Yaskawa INFORM job: SKRZYNIA_4840_-90_STOPNI_10BR.JBI

/JOB
//NAME SKRZYNIA_4840_-90_STOPNI_10BR
///FOLDERNAME 02-SKRZYNIE_JOBS
//POS
///NPOS 688,688,0,49,0,0
///TOOL 0
///POSTYPE PULSE
///PULSE
C00000=0,-52280,40443,0,6876,0
C00001=-82314,-24956,17040,-59626,-27382,-6248
C00002=-93910,-8625,17040,-59626,-43355,-6248
C00003=-98846,-1061,-42166,-80308,-57081,16120
C00004=-100452,6057,-48127,-85711,-56704,21322
C00005=-96957,25597,-37888,-85158,-62082,25522
C00006=-95580,33075,-33256,-84644,-64024,26851
C00007=-94380,33739,-32188,-85134,-63496,26721
C00008=-95580,33075,-33256,-84644,-64024,26851
C00009=-94940,31262,-36138,-85248,-63712,27160
C00010=-95580,33075,-33256,-84644,-64024,26851
C00011=-95263,33142,-33256,-84677,-63995,26850
C00012=-95263,33142,-33256,-84677,-63995,26850
C00013=-94261,33702,-32359,-85087,-63552,26740
C00014=-95263,33142,-33256,-84677,-63995,26850
C00015=-94777,31773,-35433,-85135,-63758,27084
C00016=-95263,33142,-33256,-84677,-63995,26850
C00017=-95260,33144,-33256,-84678,-63995,26850
C00018=-95260,33144,-33256,-84678,-63995,26850
C00019=-94282,33689,-32380,-85076,-63563,26742
C00020=-95260,33144,-33256,-84678,-63995,26850
C00021=-94827,31920,-35204,-85086,-63784,27059
C00022=-95260,33144,-33256,-84678,-63995,26850
C00023=-95258,33145,-33257,-84676,-63996,26846
C00024=-95258,33145,-33257,-84676,-63996,26846
C00025=-94286,33686,-32387,-85074,-63568,26738
C00026=-95258,33145,-33257,-84676,-63996,26846
C00027=-94874,32057,-34990,-85039,-63809,27032
C00028=-95258,33145,-33257,-84676,-63996,26846
C00029=-95258,33145,-33257,-84676,-63996,26846
C00030=-95258,33145,-33257,-84676,-63996,26846
C00031=-94323,33667,-32422,-85059,-63584,26741
C00032=-95258,33145,-33257,-84676,-63996,26846
C00033=-94899,32130,-34875,-85014,-63820,27019
C00034=-95258,33145,-33257,-84676,-63996,26846
C00035=-95258,25631,32269,-66559,-75499,2416
C00036=-95258,25631,32269,-66559,-75499,2416
C00037=-94333,26371,33350,-66433,-74983,2224
C00038=-95258,25631,32269,-66559,-75499,2416
C00039=-94886,24142,30119,-66602,-75133,2534
C00040=-95258,25631,32269,-66559,-75499,2416
C00041=-98646,19496,-17631,-99827,-80462,21224
C00042=-98811,21047,-15512,-99242,-81394,20987
C00043=-97886,21574,-14788,-99528,-80824,20997
C00044=-98811,21047,-15512,-99242,-81394,20987
C00045=-98517,19954,-17009,-99363,-81263,21101
C00046=-98811,21047,-15512,-99242,-81394,20987
C00047=-98811,19937,1242,-97498,-78933,15296
C00048=-98811,19937,1242,-97498,-78933,15296
C00049=-97933,20465,1962,-97646,-78345,15298
C00050=-98811,19937,1242,-97498,-78933,15296
C00051=-98523,18806,-285,-97586,-78782,15407
C00052=-98811,19937,1242,-97498,-78933,15296
C00053=-98215,26829,34899,-99955,-75775,7961
C00054=-97536,27946,37844,-102629,-75095,7996
C00055=-96676,28621,38852,-102572,-74482,7985
C00056=-97536,27946,37844,-102629,-75095,7996
C00057=-97073,25840,34734,-102750,-74944,8293
C00058=-97536,27946,37844,-102629,-75095,7996
C00059=-96761,21976,18943,-104804,-75068,12116
C00060=-92262,-3556,-2957,-107669,-51219,12798
C00061=-85502,-24407,-19904,-109451,-30096,13932
C00062=-50003,-39410,-5978,-16260,-18649,-25999
C00063=-48287,-44591,-17414,-16172,-14532,-25809
C00064=-85348,-13130,13838,-41209,-47455,-8220
C00065=-99199,18818,35660,-68259,-73735,6208
C00066=-95720,15423,18785,-70454,-68603,10022
C00067=-95720,15423,18785,-70454,-68603,10022
C00068=-97322,30100,38585,-71742,-79662,10416
C00069=-96349,30901,39804,-71630,-79090,10224
C00070=-97322,30100,38585,-71742,-79662,10416
C00071=-97054,28837,36680,-71776,-79387,10556
C00072=-97322,30100,38585,-71742,-79662,10416
C00073=-97373,30352,38967,-71736,-79717,10385
C00074=-97373,30352,38967,-71736,-79717,10385
C00075=-96432,31128,40151,-71627,-79165,10198
C00076=-97373,30352,38967,-71736,-79717,10385
C00077=-97071,28917,36802,-71776,-79407,10544
C00078=-97373,30352,38967,-71736,-79717,10385
C00079=-97356,30262,38827,-71739,-79698,10398
C00080=-97356,30262,38827,-71739,-79698,10398
C00081=-96507,30957,39891,-71642,-79201,10230
C00082=-97356,30262,38827,-71739,-79698,10398
C00083=-97092,29010,36937,-71773,-79425,10538
C00084=-97356,30262,38827,-71739,-79698,10398
C00085=-97431,30641,39402,-71725,-79780,10352
C00086=-97431,30641,39402,-71725,-79780,10352
C00087=-96578,31348,40481,-71627,-79280,10181
C00088=-97431,30641,39402,-71725,-79780,10352
C00089=-97114,29116,37095,-71767,-79448,10523
C00090=-97431,30641,39402,-71725,-79780,10352
C00091=-99948,24360,13310,-86634,-79084,-1692
C00092=-99948,24360,13310,-86634,-79084,-1692
C00093=-99080,24906,14086,-86708,-78501,-1755
C00094=-99948,24360,13310,-86634,-79084,-1692
C00095=-99633,22968,11346,-86719,-78869,-1551
C00096=-99948,24360,13310,-86634,-79084,-1692
C00097=-97019,23700,25794,-103927,-75007,-5801
C00098=-97395,30282,35552,-103352,-78262,-7023
C00099=-96588,30934,36542,-103330,-77681,-7037
C00100=-97395,30282,35552,-103352,-78262,-7023
C00101=-97049,28659,33116,-103437,-78167,-6786
C00102=-97395,30282,35552,-103352,-78262,-7023
C00103=-90014,-10558,-39023,-122472,-57861,10563
C00104=-96923,-13864,-45757,-120418,-62715,10144
C00105=-81853,-22326,-62247,-144804,-57102,19611
C00106=-90840,-27079,-68635,-139700,-60795,17408
C00107=-59535,-63832,-86313,-155973,-37716,23892
C00108=-73187,-23116,26488,-26118,-57509,-28469
C00109=-99665,-12992,-24886,-73613,-54905,-950
C00110=-98398,-8109,-25057,-81551,-55130,4513
C00111=-99451,17861,2757,-80571,-73406,6045
C00112=-99056,24650,11359,-80216,-77425,5946
C00113=-98115,25261,12228,-80295,-76818,5843
C00114=-99056,24650,11359,-80216,-77425,5946
C00115=-98800,23560,9817,-80291,-77224,6050
C00116=-99056,24650,11359,-80216,-77425,5946
C00117=-99819,33446,48735,-87787,-79679,-1235
C00118=-99819,33446,48735,-87787,-79679,-1235
C00119=-98945,34179,49898,-87659,-79086,-1350
C00120=-99819,33446,48735,-87787,-79679,-1235
C00121=-99591,32133,46677,-87830,-79529,-1033
C00122=-99819,33446,48735,-87787,-79679,-1235
C00123=-98853,28116,28355,-96898,-79749,4777
C00124=-98853,30464,37910,-96149,-78952,2546
C00125=-98284,30904,38579,-96116,-78548,2515
C00126=-98853,30464,37910,-96149,-78952,2546
C00127=-98656,29478,36421,-96191,-78865,2688
C00128=-98853,30464,37910,-96149,-78952,2546
C00129=-94437,3365,15121,-90804,-55123,21
C00130=-76606,-19838,2636,-59027,-23020,-13375
C00131=-49667,-45532,-21960,-5654,-17518,-35856
C00132=-47485,-50287,-32535,-1070,-13732,-37871
C00133=-36103,-65917,11738,-26975,4295,7905
C00134=6327,-52297,40484,-8600,6957,5944
C00135=0,-43112,23163,32261,-40956,29092
C00136=-48283,-21883,28214,-25170,-26491,48363
C00137=-46664,-3144,58041,-18842,-32105,45325
C00138=-50347,-18571,12268,-49104,-16423,60029
C00139=-53571,-17125,12073,-56866,-17385,63433
C00140=-52069,-15730,13206,-55612,-16432,62999
C00141=-53474,-15384,13495,-57637,-17161,63825
C00142=-53571,-17125,12073,-56866,-17385,63433
C00143=-50509,-19000,10610,-51503,-15997,61182
C00144=-53130,-17211,12007,-56251,-17152,63186
C00145=-51822,-15992,12994,-55136,-16324,62798
C00146=-53635,-15431,13457,-57815,-17251,63894
C00147=-53130,-17211,12007,-56251,-17152,63186
C00148=-50704,-18403,11069,-52157,-16018,61478
C00149=-53231,-16470,14622,-53206,-17893,61673
C00150=-51756,-15101,15744,-51790,-16990,61165
C00151=-53741,-14453,16285,-54808,-17949,62397
C00152=-53231,-17580,11714,-56182,-17246,63139
C00153=-51814,-19410,10295,-53186,-16720,61844
C00154=-53629,-18979,7405,-62018,-16535,65958
C00155=-52238,-17698,8415,-61175,-15613,65699
C00156=-53551,-17401,8655,-62910,-16346,66402
C00157=-52880,-17654,11656,-55678,-17066,62935
C00158=-51005,-17995,11387,-52847,-16122,61778
C00159=-52964,-17611,11689,-55811,-17106,62990
C00160=-51611,-16353,12697,-54642,-16249,62582
C00161=-53495,-15765,13180,-57466,-17201,63739
C00162=-52964,-17611,11689,-55811,-17106,62990
C00163=-51030,-17982,11395,-52891,-16135,61798
C00164=-52975,-17563,11726,-55850,-17109,63009
C00165=-51607,-16289,12749,-54669,-16241,62596
C00166=-53283,-15811,13140,-57177,-17094,63622
C00167=-52975,-17563,11726,-55850,-17109,63009
C00168=-50945,-18019,11363,-52741,-16103,61737
C00169=-52728,-17788,11545,-55393,-17010,62816
C00170=-51045,-16207,12813,-53894,-15944,62287
C00171=-52895,-15647,13274,-56746,-16874,63461
C00172=-52728,-17788,11545,-55393,-17010,62816
C00173=-50945,-18019,11363,-52741,-16103,61737
C00174=-52556,-17520,11756,-55311,-16888,62798
C00175=-51113,-16157,12849,-54025,-15975,62343
C00176=-52730,-15718,13210,-56498,-16792,63358
C00177=-52556,-17520,11756,-55311,-16888,62798
C00178=-50945,-18019,11363,-52741,-16103,61737
C00179=-51893,-17787,11546,-54246,-16568,62356
C00180=-50379,-16341,12703,-52826,-15610,61849
C00181=-52406,-15704,13225,-56071,-16614,63190
C00182=-51893,-17787,11546,-54246,-16568,62356
C00183=-50028,-22953,-3957,-22347,-31919,54220
C00184=-50947,-22502,-3625,-23433,-32061,54736
C00185=-49421,-20951,-2455,-21951,-31329,54057
C00186=-51207,-20433,-2055,-24026,-31698,55041
C00187=-50529,-22709,-3778,-22940,-31995,54502
C00188=-49763,-25421,-36239,-24565,-26935,60445
C00189=-49763,-25421,-36239,-24565,-26935,60445
C00190=-48299,-23485,-34758,-23276,-26122,59713
C00191=-50218,-22723,-34165,-25568,-26529,60993
C00192=-49763,-25421,-36239,-24565,-26935,60445
C00193=-50713,-12366,-58367,-41124,-17813,74400
C00194=-50824,-12254,-58263,-41255,-17847,74484
C00195=-49431,-10052,-56192,-40383,-17131,73813
C00196=-50915,-9358,-55524,-41955,-17664,74847
C00197=-51028,-12852,-58814,-41301,-17980,74542
C00198=-49763,-25421,-36239,-24565,-26935,60445
C00199=-50529,-22709,-3778,-22940,-31995,54502
C00200=-45389,-28224,4312,-35967,-15579,54278
C00201=-40154,-51179,-915,-24203,-8234,36524
C00202=0,-52280,40443,0,6876,0
C00203=0,-52280,40443,0,6876,0
C00204=-2117,-50103,-33543,-4117,45077,85249
C00205=26439,-48928,-33543,-4117,-52362,85249
C00206=26439,-27355,-33543,-41485,-52362,85249
C00207=39218,-24492,-41653,-51934,-39374,86964
C00208=39218,-24492,-41653,-51934,-39374,86964
C00209=46639,7575,-9331,-26045,-41627,82486
C00210=47278,8641,-9483,-26175,-40625,82510
C00211=46369,10567,-7126,-26545,-41054,82831
C00212=47278,8641,-9483,-26175,-40625,82510
C00213=48256,9506,-8430,-25641,-40400,82076
C00214=47278,8641,-9483,-26175,-40625,82510
C00215=44522,-635,-31983,-49264,-28311,89687
C00216=44247,-628,-31975,-49394,-28443,89790
C00217=43310,1314,-29842,-49807,-28910,90140
C00218=44247,-628,-31975,-49394,-28443,89790
C00219=45313,152,-31124,-48894,-27920,89380
C00220=44247,-628,-31975,-49394,-28443,89790
C00221=41572,-13073,-22520,-50760,-38355,84033
C00222=21909,-6773,-14577,-94161,-56302,89381
C00223=23773,-3183,-10897,-94486,-55065,89563
C00224=24904,-823,-8382,-94654,-54308,89644
C00225=24395,1151,-6219,-94590,-54651,89617
C00226=24904,-823,-8382,-94654,-54308,89644
C00227=26178,-337,-7854,-94816,-53451,89710
C00228=24904,-823,-8382,-94654,-54308,89644
C00229=17020,-16061,-23281,-93084,-59494,88637
C00230=-21568,-26506,-31664,-90508,-85573,86639
C00231=-8557,-39769,-22319,-51419,-69406,84680
C00232=-8557,-39769,-22319,-51419,-69406,84680
C00233=32994,-9735,-10751,-29019,-59471,69498
C00234=43974,9628,-22604,-36190,-36396,73426
C00235=45932,13115,-22315,-37472,-33732,73846
C00236=45228,14664,-20329,-37571,-34159,74020
C00237=45932,13115,-22315,-37472,-33732,73846
C00238=46653,13731,-21526,-37109,-33514,73520
C00239=45932,13115,-22315,-37472,-33732,73846
C00240=39039,866,-6986,-42761,-44691,67687
C00241=30717,-9248,-22721,-77433,-42696,79486
C00242=32434,-7077,-20587,-77571,-41526,79457
C00243=31883,-5576,-19073,-77676,-41878,79560
C00244=32434,-7077,-20587,-77571,-41526,79457
C00245=33092,-6769,-20280,-77576,-41084,79417
C00246=32434,-7077,-20587,-77571,-41526,79457
C00247=30527,-14106,-27266,-76898,-42917,79150
C00248=25454,-9581,-17335,-94425,-53880,89429
C00249=24965,-2445,-10120,-94645,-54263,89631
C00250=24893,-1278,-8874,-94650,-54314,89639
C00251=24417,557,-6877,-94595,-54636,89618
C00252=24893,-1278,-8874,-94650,-54314,89639
C00253=25752,-956,-8526,-94759,-53737,89684
C00254=24893,-1278,-8874,-94650,-54314,89639
C00255=23817,-1527,-9142,-94518,-55040,89587
C00256=24871,-1152,-8735,-94651,-54328,89643
C00257=24440,508,-6926,-94601,-54619,89624
C00258=24871,-1152,-8735,-94651,-54328,89643
C00259=25635,-865,-8427,-94748,-53815,89684
C00260=24871,-1152,-8735,-94651,-54328,89643
C00261=33203,-4295,-13750,-123758,-49995,81034
C00262=35028,4195,-6818,-132965,-58836,87950
C00263=35028,4195,-6818,-132965,-58836,87950
C00264=34452,5837,-4911,-132720,-59045,87770
C00265=35028,4195,-6818,-132965,-58836,87950
C00266=35710,4593,-6360,-133217,-58512,88125
C00267=35028,4195,-6818,-132965,-58836,87950
C00268=24762,-11408,-28656,-113055,-60293,85383
C00269=-28645,-26349,-41223,-103369,-91870,78302
C00270=-28645,-26349,-41223,-103369,-91870,78302
C00271=-25549,-24286,-26215,-66769,-87032,80148
C00272=27561,-8271,-12315,-63268,-52553,74387
C00273=29336,-165,-3925,-63163,-51316,74265
C00274=29518,765,-2904,-63127,-51205,74233
C00275=28850,2962,-447,-63227,-51636,74327
C00276=29518,765,-2904,-63127,-51205,74233
C00277=30662,1292,-2320,-62902,-50501,74035
C00278=29518,765,-2904,-63127,-51205,74233
C00279=30773,10953,32136,-106912,-46141,83783
C00280=30773,10953,32136,-106912,-46141,83783
C00281=30080,13410,35293,-106601,-46463,83481
C00282=30773,10953,32136,-106912,-46141,83783
C00283=32007,11622,32987,-106899,-45346,83915
C00284=30773,10953,32136,-106912,-46141,83783
C00285=28321,-8642,-16372,-95739,-47180,89965
C00286=28583,-7344,-15096,-95864,-47019,90043
C00287=27897,-5229,-12965,-95873,-47499,90079
C00288=28583,-7344,-15096,-95864,-47019,90043
C00289=29900,-6813,-14567,-96101,-46141,90154
C00290=28583,-7344,-15096,-95864,-47019,90043
C00291=27852,-7537,-15286,-95742,-47508,89986
C00292=28448,-7306,-15058,-95845,-47110,90035
C00293=27795,-5283,-13021,-95851,-47567,90065
C00294=28448,-7306,-15058,-95845,-47110,90035
C00295=29772,-6774,-14527,-96083,-46226,90146
C00296=28448,-7306,-15058,-95845,-47110,90035
C00297=18552,-19531,-26179,-93438,-53589,88597
C00298=40301,-14999,-52277,-148979,-69262,86714
C00299=42323,-33,-37432,-150113,-69667,87489
C00300=53245,19091,3515,-165691,-72595,90030
C00301=53641,19552,4138,-165817,-72473,90151
C00302=53058,20743,5761,-165615,-72317,89948
C00303=53641,19552,4138,-165817,-72473,90151
C00304=54155,20160,4967,-165982,-72308,90306
C00305=53641,19552,4138,-165817,-72473,90151
C00306=23439,-10154,-17205,-109204,-58547,76547
C00307=2382,-21913,-40813,-107544,-74451,77239
C00308=-31257,-15877,-35733,-102288,-96107,74463
C00309=-39204,-18003,-7668,-86141,-99190,68413
C00310=-5592,-5690,18047,-75373,-79525,63129
C00311=19039,-439,25862,-68224,-64120,61443
C00312=21624,5223,26011,-69375,-61155,63193
C00313=24437,11840,34139,-68260,-59598,62567
C00314=24053,13588,36402,-68249,-59917,62491
C00315=24437,11840,34139,-68260,-59598,62567
C00316=25079,12112,34488,-68051,-59212,62472
C00317=24437,11840,34139,-68260,-59598,62567
C00318=21370,4935,25667,-69451,-61310,63230
C00319=-18351,-11002,3811,-80352,-86206,66275
C00320=-34619,-5846,8788,-82342,-97004,67025
C00321=-40684,-19963,-8478,-86482,-100204,67987
C00322=1570,-13136,-5998,-86227,-71173,69099
C00323=13966,-6596,-2340,-86587,-62612,70052
C00324=24093,-1862,-9504,-94546,-54850,89594
C00325=24093,-1862,-9504,-94546,-54850,89594
C00326=23519,425,-7024,-94488,-55240,89573
C00327=24093,-1862,-9504,-94546,-54850,89594
C00328=25256,-1442,-9053,-94693,-54067,89656
C00329=24093,-1862,-9504,-94546,-54850,89594
C00330=27718,4364,12871,-105518,-51077,86669
C00331=27718,4364,12871,-105518,-51077,86669
C00332=27164,6353,15202,-105385,-51398,86539
C00333=27718,4364,12871,-105518,-51077,86669
C00334=28828,4851,13441,-105618,-50355,86801
C00335=27718,4364,12871,-105518,-51077,86669
C00336=20930,-1364,27707,-95004,-52134,77785
C00337=-41463,-32191,18163,-91991,-64949,55938
C00338=0,-52277,40442,0,6872,4
C00339=-82314,-24956,17040,-59626,-27382,-6248
C00340=-93910,-8625,17040,-59626,-43355,-6248
C00341=-98846,-1061,-42166,-80308,-57081,16120
C00342=-100452,6057,-48127,-85711,-56704,21322
C00343=-95564,34698,-34234,-85516,-63941,27819
C00344=-94221,34299,-28769,-82558,-65564,25844
C00345=-94107,37241,-30442,-84005,-65307,27544
C00346=-95103,32620,-31323,-83378,-64939,26072
C00347=-95103,32620,-31323,-83378,-64939,26072
C00348=-93990,32828,-31380,-83932,-64473,26160
C00349=-94063,31710,-30585,-83283,-64598,25457
C00350=-96692,32939,-31211,-82617,-65723,26190
C00351=-96111,21840,170,-71736,-70232,11396
C00352=-94229,22391,773,-71789,-70557,11468
C00353=-94283,22521,1025,-71678,-70686,11433
C00354=-95675,19167,-4176,-72970,-68231,11735
C00355=-95681,24338,3488,-71459,-71669,11415
C00356=-94245,22750,1246,-71757,-70674,11453
C00357=-94341,22923,1499,-71729,-70746,11440
C00358=-96213,24222,3324,-71394,-71999,11479
C00359=-95517,23330,2066,-71543,-71508,11507
C00360=-94304,22892,1449,-71738,-70721,11443
C00361=-94158,22889,1452,-71756,-70627,11429
C00362=-96071,24319,3461,-71408,-71916,11455
C00363=-96941,-6406,-33809,-76117,-54125,10511
C00364=-90643,-26862,-25633,-62597,-56791,-1368
C00365=-66103,-61757,7450,-21008,-32955,-5749
C00366=4223,-52290,40457,-5766,6913,3980
C00367=4223,-52290,40457,-5766,6913,3980
C00368=-4538,-50065,-33535,-3011,44998,84219
C00369=24207,-49248,-33668,-5551,-52644,86091
C00370=25094,-27722,-33812,-41887,-53054,85599
C00371=38036,-25052,-42086,-52219,-40087,87228
C00372=37328,-2824,-24733,-57182,-37821,90318
C00373=36700,-2520,-13735,-51589,-42201,86442
C00374=37520,2330,-3498,-48550,-43875,84431
C00375=37520,1020,-12079,-52650,-40851,87066
C00376=48458,-261,-12985,-24069,-43340,80504
C00377=36153,7296,-1758,-40139,-50302,89334
C00378=37146,11264,2520,-40849,-50296,89553
C00379=38059,11410,-1863,-40565,-47910,90206
C00380=36726,6476,-7858,-41213,-48206,90783
C00381=19339,7883,9818,-77509,-64249,74140
C00382=19027,1888,-16187,-103553,-67480,82955
C00383=24158,3537,-14322,-106039,-60939,84018
C00384=24143,4321,-7309,-103852,-59670,81875
C00385=19531,2904,-8928,-102027,-65985,80961
C00386=20232,-3383,-14682,-86495,-63009,78978
C00387=-24375,-51634,-49601,-83793,-94064,73950
C00388=4223,-52290,40457,-5766,6913,3980
C00389=-4825,-36686,24602,37792,-30278,35378
C00390=-46221,-29633,7403,-27051,-24124,46751
C00391=-46221,-29633,7403,-27051,-24124,46751
C00392=-52474,-20611,11454,-41004,-23045,52959
C00393=-60257,-19980,-2088,-84190,-23320,82051
C00394=-63868,-19883,-6318,-95759,-28031,88346
C00395=-51819,-22965,8574,-41365,-22900,53139
C00396=-4825,-36686,24602,37792,-30278,35378
C00397=0,-52280,40443,0,6876,0
C00398=4223,-52290,40457,-5766,6913,3980
C00399=-66103,-61757,7450,-21008,-32955,-5749
C00400=-89093,-33107,-44597,-67545,-52550,2722
C00401=-96941,-6406,-33809,-76117,-54125,10511
C00402=-99429,14378,84,-80785,-71596,8628
C00403=-99699,24313,24829,-82602,-77917,4569
C00404=-98066,26841,20697,-83331,-79245,6860
C00405=-98079,26929,20513,-83349,-79351,6953
C00406=-99638,19663,10292,-84193,-74452,7551
C00407=-99636,19665,10291,-84197,-74448,7550
C00408=-98131,26698,20177,-83371,-79212,6975
C00409=-98097,25980,12653,-84102,-79057,9159
C00410=-99636,19665,10291,-84197,-74448,7550
C00411=-99898,19397,9265,-91157,-75555,8932
C00412=-98443,26671,19736,-90040,-80194,8298
C00413=-98497,26824,19963,-90017,-80321,8279
C00414=-99898,19397,9265,-91157,-75555,8932
C00415=-100050,15245,3951,-91671,-73354,9137
C00416=-100612,486,21817,-80549,-57848,-3680
C00417=-100400,-9442,6808,-74817,-59142,-3019
C00418=-61441,-38616,11032,-55510,-42874,-3049
C00419=4223,-52290,40457,-5766,6913,3980
C00420=-22331,-23394,-30093,-82917,-82006,85712
C00421=22434,-14401,-3235,-51104,-60845,74728
C00422=42744,21307,45077,-24753,-69813,65333
C00423=33655,14083,18147,-45417,-58301,71861
C00424=33641,11943,8279,-47835,-54840,73983
C00425=36574,13250,23432,-35354,-61822,69159
C00426=28497,326,20939,-70981,-47632,72427
C00427=30972,5983,29862,-68494,-46670,70994
C00428=31029,11571,45127,-63398,-49004,67378
C00429=28971,8096,39948,-65070,-49810,68216
C00430=29759,-12862,-24221,-91747,-41905,86600
C00431=35278,-10419,-21940,-93284,-36771,87139
C00432=36208,-10883,-22374,-93618,-35345,87231
C00433=27219,-23595,-33313,-89555,-43517,85303
C00434=10564,-40773,-45889,-85382,-54876,82708
C00435=-14984,-61618,-24572,-87392,-53367,60735
C00436=9346,-67436,-18786,-75708,-34590,53709
C00437=40938,-55232,35946,-9746,5421,6718
C00438=4223,-52290,40457,-5766,6913,3980
C00439=-4825,-36686,24602,37792,-30278,35378
C00440=-46221,-29633,7403,-27051,-24124,46751
C00441=-56796,-22932,368,-68953,-21567,70907
C00442=-61611,-20349,-6598,-95791,-25091,88405
C00443=-63740,-19715,-7390,-98604,-28245,90373
C00444=-57732,702,39416,-95701,-20291,84895
C00445=-64194,-702,47618,-60039,-31852,69283
C00446=-55070,-19477,14263,-47544,-24334,57575
C00447=-49294,-34086,9663,-30689,-30758,52546
C00448=4223,-52290,40457,-5766,6913,3980
C00449=0,-52280,40443,0,6876,0
C00450=0,-52280,40443,0,6876,0
C00451=-61754,-61602,7279,-16215,-32140,-7126
C00452=-89313,-24027,20291,-53466,-58905,-4975
C00453=-97807,-25409,-21837,-78881,-62828,2121
C00454=-95644,-21015,-18476,-76474,-46020,1039
C00455=-99748,19928,10876,-84091,-74310,7444
C00456=-97024,20398,6537,-109543,-78256,12844
C00457=-94147,25923,17140,-111429,-80132,11834
C00458=-93181,27051,21323,-113663,-79363,11504
C00459=-95358,19434,-1507,-115915,-81093,16065
C00460=-97685,-18005,-56170,-117036,-60417,20552
C00461=-60891,-56927,-71252,-134309,-22621,24600
C00462=-76377,-16480,33969,-44898,-47258,-26858
C00463=-76377,-16480,33969,-44898,-47258,-26858
C00464=-97282,11923,63589,-59034,-55972,-22399
C00465=-97282,-18199,-24804,-89107,-46272,-346
C00466=-84714,-13514,-21320,-79690,-37366,-2300
C00467=-92093,-5454,-13554,-80916,-52292,-613
C00468=-99761,24721,23429,-79408,-77929,-316
C00469=-99564,24916,23930,-79374,-77823,-417
C00470=-100005,27069,23687,-81767,-79755,895
C00471=-97295,30454,38512,-73622,-79542,-3831
C00472=-98471,27958,25022,-81751,-79627,782
C00473=-99805,23386,18402,-82055,-77455,1200
C00474=-100093,24719,20298,-81968,-77939,1081
C00475=-98451,26404,20171,-83400,-79044,-389
C00476=-98528,26732,19657,-84000,-79459,-654
C00477=-100109,23919,19160,-82044,-77303,1139
C00478=-98037,-4340,-16930,-86109,-58746,2389
C00479=-93345,-31758,-40240,-83703,-37467,-946
C00480=-81087,-35886,-14825,-53529,-36311,-18004
C00481=-47029,-49867,-20464,-11808,-29290,-36568
C00482=-41431,-67449,10869,-1325,127,-6150
C00483=6328,-52297,40483,-8599,6957,5944
C00484=-8648,-69005,-18270,-84275,-43232,53472
C00485=18757,-59462,-34892,-84638,-37529,67311
C00486=26772,-23733,-33422,-89486,-43820,85275
C00487=29039,-10071,-21608,-91386,-45181,86629
C00488=29639,-5923,-17523,-91591,-45648,86808
C00489=29709,-5453,-17046,-91618,-45636,86826
C00490=29138,-10182,-21714,-91372,-45196,86624
C00491=20424,-22725,-32635,-88800,-51006,85261
C00492=28416,-11420,-25238,-98178,-46636,84572
C00493=30481,-6584,-16425,-92636,-44382,82541
C00494=30464,-7521,-23523,-96665,-44944,85234
C00495=28416,-11420,-25238,-98178,-46636,84572
C00496=-23524,-33387,-42654,-89891,-81168,80229
C00497=-23524,-33387,-42654,-89891,-81168,80229
C00498=33935,-6399,-10013,-60506,-43064,77980
C00499=34878,-3211,-6740,-60356,-42422,77865
C00500=34873,-3218,-6748,-60357,-42424,77868
C00501=33935,-6399,-10013,-60506,-43064,77980
C00502=17782,-19597,1250,-60925,-51448,69151
C00503=-243,-43047,-13224,-69794,-55957,65877
C00504=42700,-55269,36176,-13619,5333,9062
C00505=6328,-52297,40483,-8599,6957,5944
C00506=-10231,-60460,6271,71658,-11927,-13637
C00507=-49129,-39322,3023,-34904,-18609,43900
C00508=-57258,-19535,13114,-46502,-25798,55150
C00509=-58736,-19151,1344,-78268,-22199,76919
C00510=-56868,-17231,8572,-62431,-21728,66645
C00511=-56011,-29317,6725,-41009,-27363,52457
C00512=-10137,-60963,4526,62308,-14518,-6745
C00513=0,-52280,40443,0,6876,0
C00514=0,-52280,40443,0,6876,0
C00515=-41653,-63035,2931,-3578,-7576,-14589
C00516=-45770,-50109,-20524,-10089,-29273,-37310
C00517=-80544,-36303,-15042,-52975,-36116,-18265
C00518=-93028,-32302,-40599,-83495,-37263,-1079
C00519=-98446,-3141,-15678,-86094,-59021,2414
C00520=-99951,24070,19376,-82000,-77829,1145
C00521=-98655,27908,24922,-81730,-79774,792
C00522=-98593,28720,26118,-81685,-80145,709
C00523=-99951,24070,19376,-82000,-77829,1145
C00524=-99951,24070,19376,-82000,-77829,1145
C00525=-98577,27118,23759,-81796,-79157,859
C00526=-98518,28577,26461,-81649,-79882,537
C00527=-99951,24070,19376,-82000,-77829,1145
C00528=-100269,22168,6337,-90046,-78798,5829
C00529=-98793,24504,9703,-89745,-79501,5648
C00530=-98964,25807,12446,-89411,-80347,5248
C00531=-100269,22168,6337,-90046,-78798,5829
C00532=-97981,-2707,-24332,-95437,-62441,6897
C00533=-100473,-17939,-38802,-96739,-55527,6139
C00534=-88098,-29848,-22776,-71580,-48483,-7812
C00535=-81694,-37220,-20464,-64791,-45723,-12569
C00536=-45770,-50109,-20524,-10089,-29273,-37310
C00537=-40984,-65135,6743,-2520,-4051,-10897
C00538=0,-52280,40443,0,6876,0
C00539=40939,-55232,35946,-9746,5421,6719
C00540=8707,-69002,-18268,-75213,-34271,52581
C00541=23267,-58917,-25142,-81990,-31707,62852
C00542=27307,-5613,10331,-81857,-46454,76095
C00543=30064,-5598,-963,-91827,-44222,81590
C00544=30419,-1725,5291,-88668,-43977,80354
C00545=30554,-300,10432,-88528,-43656,79164
C00546=29815,-6351,-3652,-90193,-44535,81892
C00547=29567,1847,27834,-65726,-48411,69959
C00548=23257,11670,30420,-81328,-57342,77033
C00549=23257,16856,45442,-77525,-58254,73578
C00550=21577,7912,33836,-78698,-59121,74340
C00551=17856,-9033,24892,-70658,-55966,67475
C00552=20838,-7097,2019,-111788,-62648,79114
C00553=40635,280,-7982,-142398,-56681,90238
C00554=32653,-9455,434,-90251,-40347,77213
C00555=40635,572,-6271,-142064,-55879,89947
C00556=40665,7761,2001,-141975,-55632,89869
C00557=40707,9678,10648,-140211,-51894,88431
C00558=39416,1907,3178,-139370,-51839,87774
C00559=7767,-21333,-19174,-120411,-69473,77116
C00560=33666,-18553,20064,-54519,-41956,59729
C00561=4032,-43511,13506,-33366,-30942,40837
C00562=22997,-56875,21315,16958,-8102,3163
C00563=0,-52280,40443,0,6876,0
C00564=-50974,-46557,23391,-77768,-13896,42026
C00565=-53474,-39983,4253,-39182,-18848,44272
C00566=-56619,-19856,12878,-45665,-25558,54806
C00567=-53298,-26712,-11188,-26889,-32979,52528
C00568=-57200,-20845,-7559,-37425,-33513,53351
C00569=-58648,-23818,-25853,-45100,-31207,62168
C00570=-58477,-22145,-38977,-48305,-29254,64725
C00571=-51868,-27423,-11673,-25269,-32728,51737
C00572=-49121,-45409,-2608,-26656,-19965,38583
C00573=-21301,-61008,4568,43957,-10534,-712
C00574=0,-52280,40443,0,6876,0
C00575=0,-52280,40443,0,6876,0
C00576=-40221,-67507,11044,-1325,-65,-6716
C00577=-45770,-50109,-20525,-10088,-29274,-37311
C00578=-80544,-36303,-15042,-52975,-36116,-18265
C00579=-93028,-32301,-40599,-83495,-37262,-1079
C00580=-97841,-4898,-17503,-86112,-58614,2374
C00581=-98519,20938,24576,-104669,-74039,3184
C00582=-96245,27524,33987,-104248,-75557,2188
C00583=-96042,30429,38367,-104052,-76584,1622
C00584=-98519,20938,24576,-104669,-74039,3184
C00585=-96493,25523,39222,-108744,-70575,1504
C00586=-94270,36759,56791,-107990,-72762,-811
C00587=-93688,41643,69337,-108330,-70485,-2582
C00588=-97583,22292,26930,-109533,-72865,4016
C00589=-96138,8400,8287,-106256,-65362,5540
C00590=-100287,-1716,-10146,-108305,-65235,8162
C00591=-99412,-15498,-11084,-95783,-55633,1327
C00592=-91712,-24690,-5004,-66532,-53484,-12011
C00593=-45770,-50109,-20525,-10088,-29274,-37311
C00594=-40221,-67507,11044,-1325,-65,-6716
C00595=0,-52280,40443,0,6876,0
C00596=51241,-30653,28678,4016,-29070,6398
C00597=46185,-61941,-37286,-12736,-10732,51851
C00598=-13205,-44768,-23966,-65315,-59418,73750
C00599=-11120,-40541,-20876,-69249,-61539,75403
C00600=-836,-13033,12361,-83908,-73576,73378
C00601=18912,6214,32354,-79489,-60743,73080
C00602=21217,10898,38129,-78632,-59343,72736
C00603=23447,16313,45262,-77527,-58074,72177
C00604=23610,23756,64158,-73325,-59549,68283
C00605=18912,6214,32354,-79489,-60743,73080
C00606=-836,-13033,12361,-83908,-73576,73378
C00607=-20209,-39682,-20467,-71924,-67122,76479
C00608=-20209,-39682,-20467,-71924,-67122,76479
C00609=26353,-3691,11741,-61723,-54035,71160
C00610=29598,-2090,11073,-69087,-47235,76987
C00611=30217,-1844,4641,-75777,-45517,79979
C00612=29529,1742,11379,-68166,-49318,73572
C00613=24010,-9039,-4437,-79986,-50972,77255
C00614=24652,-10740,-12845,-99298,-50700,81949
C00615=28976,-2672,-4778,-100308,-47937,82653
C00616=31030,-2921,-9996,-112394,-49006,86348
C00617=24652,-10740,-12845,-99298,-50700,81949
C00618=-25637,-26222,-38592,-96633,-85474,81576
C00619=-36771,-16470,-4689,-95304,-89579,74076
C00620=-33704,-12343,7746,-85568,-87064,70052
C00621=4032,-43511,13506,-33366,-30942,40837
C00622=27500,-60047,23168,28912,-2679,-5784
C00623=0,-52280,40443,0,6876,0
C00624=-50971,-46557,23390,-77766,-13895,42026
C00625=-53475,-39984,4253,-39182,-18848,44273
C00626=-56619,-19856,12878,-45665,-25558,54806
C00627=-57643,-27958,-8553,-51854,-24771,59787
C00628=-66195,-24410,-19095,-90567,-31132,85904
C00629=-63290,-24193,-14362,-80030,-27547,78073
C00630=-39040,-40975,-15408,-18643,-21575,44866
C00631=-11647,-69843,-10959,56399,-11165,-4616
C00632=-15394,-57237,30542,-10392,5525,8219
C00633=0,-52280,40443,0,6876,0
C00634=0,-52280,40443,0,6876,0
C00635=-40221,-67507,11044,-1325,-65,-6716
C00636=-45770,-50109,-20525,-10088,-29274,-37311
C00637=-95022,-19559,-3970,-66108,-42168,-11789
C00638=-84972,-7110,7117,-67721,-41324,-10731
C00639=-83869,-8155,6098,-67213,-40658,-10968
C00640=-99927,23961,20220,-85683,-78298,772
C00641=-98562,26853,28284,-85090,-78334,-823
C00642=-98562,24944,18750,-86001,-78172,1594
C00643=-99839,23064,19027,-85806,-76881,822
C00644=-99837,28317,40379,-83872,-77348,-4229
C00645=-98320,27099,26117,-95522,-79020,1523
C00646=-98352,30753,38436,-94609,-78846,-1184
C00647=-98854,25297,30332,-94828,-76302,-321
C00648=-96904,30940,39860,-101743,-77102,-265
C00649=-96724,33273,50535,-100476,-74766,-2729
C00650=-98804,25282,29667,-102283,-76702,1142
C00651=-100571,27242,38707,-91767,-77267,-2786
C00652=-98525,26014,33005,-89185,-76389,-1063
C00653=-98525,23467,22318,-90325,-76630,1518
C00654=-99839,23064,19027,-85806,-76881,822
C00655=-86774,-13232,-16630,-85484,-41019,-1154
C00656=-97999,-21060,-29835,-88214,-48653,956
C00657=-98846,-3268,25064,-74217,-51189,-12584
C00658=-70313,-35289,-4922,-51188,-38634,-20596
C00659=-81694,-37221,-20464,-64791,-45723,-12569
C00660=-45770,-50109,-20525,-10088,-29274,-37311
C00661=-41628,-63095,3038,-3547,-7472,-14475
C00662=4224,-52288,40457,-5773,6909,3978
C00663=4224,-52288,40457,-28770,-64753,45638
C00664=6548,2882,44080,-77825,-67624,70557
C00665=22702,21750,69443,-66118,-61597,67582
C00666=25585,21999,63350,-62249,-61285,68688
C00667=25777,17209,50811,-62979,-59886,70957
C00668=23226,22825,71113,-65575,-61542,67353
C00669=24931,14697,51677,-80718,-51653,72069
C00670=24746,14409,39758,-87518,-53542,76879
C00671=24784,21556,58944,-82031,-53873,72431
C00672=22657,12722,42993,-85587,-54940,74916
C00673=-4427,-20395,-7318,-104668,-69521,79317
C00674=768,-20151,-3587,-97758,-65802,76626
C00675=-14736,-21545,-1233,-93598,-60476,72578
C00676=1642,-46684,14475,-47609,-24983,34912
C00677=27500,-60047,23168,28912,-2679,-5784
C00678=0,-52280,40443,0,6876,0
C00679=-50971,-46557,23390,-77766,-13895,42026
C00680=-53475,-39984,4253,-39182,-18848,44273
C00681=-56619,-19856,12878,-45665,-25558,54806
C00682=-53891,-17708,14512,-43170,-23995,53902
C00683=-60674,-17500,6427,-71116,-24772,71097
C00684=-63181,-17997,2063,-82122,-26831,78394
C00685=-39402,-27697,7664,-17904,-21663,43170
C00686=-11647,-69843,-10959,56399,-11165,-4616
C00687=0,-52280,40443,0,6876,0
BC00000=464364
BC00001=445130
BC00002=445130
BC00003=445130
BC00004=445130
BC00005=445130
BC00006=445130
BC00007=445130
BC00008=445130
BC00009=445130
BC00010=445130
BC00011=491232
BC00012=491232
BC00013=491232
BC00014=491232
BC00015=491232
BC00016=491232
BC00017=537442
BC00018=537442
BC00019=537442
BC00020=537442
BC00021=537442
BC00022=537442
BC00023=583546
BC00024=583546
BC00025=583546
BC00026=583546
BC00027=583546
BC00028=583546
BC00029=606594
BC00030=606594
BC00031=606594
BC00032=606594
BC00033=606594
BC00034=606594
BC00035=559393
BC00036=559393
BC00037=559393
BC00038=559393
BC00039=559393
BC00040=559393
BC00041=605503
BC00042=605503
BC00043=605504
BC00044=605503
BC00045=605503
BC00046=605503
BC00047=605503
BC00048=605503
BC00049=605503
BC00050=605503
BC00051=605503
BC00052=605503
BC00053=598111
BC00054=596575
BC00055=596575
BC00056=596575
BC00057=596575
BC00058=596575
BC00059=601183
BC00060=585822
BC00061=564496
BC00062=564906
BC00063=699121
BC00064=714117
BC00065=714117
BC00066=714117
BC00067=714117
BC00068=714117
BC00069=714117
BC00070=714117
BC00071=714117
BC00072=714117
BC00073=737203
BC00074=737203
BC00075=737203
BC00076=737203
BC00077=737203
BC00078=737203
BC00079=783275
BC00080=783275
BC00081=783275
BC00082=783275
BC00083=783275
BC00084=783275
BC00085=806364
BC00086=806364
BC00087=806364
BC00088=806364
BC00089=806364
BC00090=806364
BC00091=841654
BC00092=841654
BC00093=841654
BC00094=841654
BC00095=841654
BC00096=841654
BC00097=835379
BC00098=835379
BC00099=835379
BC00100=835379
BC00101=835379
BC00102=835379
BC00103=847091
BC00104=848363
BC00105=846315
BC00106=845191
BC00107=849235
BC00108=914118
BC00109=954480
BC00110=945981
BC00111=946006
BC00112=946012
BC00113=946012
BC00114=946012
BC00115=946012
BC00116=946012
BC00117=942336
BC00118=942336
BC00119=942336
BC00120=942336
BC00121=942336
BC00122=942336
BC00123=957753
BC00124=957753
BC00125=957753
BC00126=957753
BC00127=957753
BC00128=957753
BC00129=940598
BC00130=924233
BC00131=927607
BC00132=905277
BC00133=834851
BC00134=786663
BC00135=811795
BC00136=904340
BC00137=904340
BC00138=933642
BC00139=935739
BC00140=935739
BC00141=935739
BC00142=935739
BC00143=889624
BC00144=889624
BC00145=889624
BC00146=889624
BC00147=889624
BC00148=828182
BC00149=828182
BC00150=828182
BC00151=828182
BC00152=828182
BC00153=766752
BC00154=766752
BC00155=766752
BC00156=766752
BC00157=766752
BC00158=705350
BC00159=705350
BC00160=705350
BC00161=705350
BC00162=705350
BC00163=643865
BC00164=643865
BC00165=643865
BC00166=643865
BC00167=643865
BC00168=582464
BC00169=582464
BC00170=582464
BC00171=582464
BC00172=582464
BC00173=520992
BC00174=520992
BC00175=520992
BC00176=520992
BC00177=520992
BC00178=459540
BC00179=459540
BC00180=459540
BC00181=459540
BC00182=459540
BC00183=459544
BC00184=459544
BC00185=459544
BC00186=459544
BC00187=459544
BC00188=459544
BC00189=459544
BC00190=459544
BC00191=459544
BC00192=459544
BC00193=459544
BC00194=459544
BC00195=459544
BC00196=459544
BC00197=459544
BC00198=459544
BC00199=459544
BC00200=459540
BC00201=533216
BC00202=533216
BC00203=492150
BC00204=423885
BC00205=423885
BC00206=423885
BC00207=423885
BC00208=423885
BC00209=493160
BC00210=493160
BC00211=493160
BC00212=493160
BC00213=493160
BC00214=493160
BC00215=539180
BC00216=539180
BC00217=539180
BC00218=539180
BC00219=539180
BC00220=539180
BC00221=525487
BC00222=485388
BC00223=485386
BC00224=485384
BC00225=485384
BC00226=485384
BC00227=485384
BC00228=485384
BC00229=485384
BC00230=485384
BC00231=485384
BC00232=635507
BC00233=635507
BC00234=635507
BC00235=635509
BC00236=635509
BC00237=635509
BC00238=635509
BC00239=635509
BC00240=603035
BC00241=594948
BC00242=594948
BC00243=594948
BC00244=594948
BC00245=594948
BC00246=594948
BC00247=594948
BC00248=600591
BC00249=600589
BC00250=600589
BC00251=600589
BC00252=600589
BC00253=600589
BC00254=600589
BC00255=623637
BC00256=623637
BC00257=623637
BC00258=623637
BC00259=623637
BC00260=623637
BC00261=623637
BC00262=623637
BC00263=623637
BC00264=623637
BC00265=623637
BC00266=623637
BC00267=623637
BC00268=623637
BC00269=623637
BC00270=758391
BC00271=758391
BC00272=758391
BC00273=758391
BC00274=758391
BC00275=758391
BC00276=758391
BC00277=758391
BC00278=758391
BC00279=669704
BC00280=669704
BC00281=669706
BC00282=669704
BC00283=669704
BC00284=669704
BC00285=784942
BC00286=784942
BC00287=784942
BC00288=784942
BC00289=784942
BC00290=784942
BC00291=807985
BC00292=807985
BC00293=807985
BC00294=807985
BC00295=807985
BC00296=807985
BC00297=807985
BC00298=784942
BC00299=784942
BC00300=784942
BC00301=784942
BC00302=784942
BC00303=784942
BC00304=784942
BC00305=784942
BC00306=785203
BC00307=785203
BC00308=785203
BC00309=895226
BC00310=895226
BC00311=895226
BC00312=895226
BC00313=895226
BC00314=895226
BC00315=895226
BC00316=895226
BC00317=895226
BC00318=895226
BC00319=906894
BC00320=906894
BC00321=963281
BC00322=963281
BC00323=963281
BC00324=969297
BC00325=969297
BC00326=969297
BC00327=969297
BC00328=969297
BC00329=969297
BC00330=969297
BC00331=969297
BC00332=969297
BC00333=969297
BC00334=969297
BC00335=969297
BC00336=927243
BC00337=883644
BC00338=475149
BC00339=445130
BC00340=445130
BC00341=445130
BC00342=445130
BC00343=445130
BC00344=445710
BC00345=445126
BC00346=445722
BC00347=484130
BC00348=492177
BC00349=481766
BC00350=492273
BC00351=473247
BC00352=480563
BC00353=473247
BC00354=480984
BC00355=519338
BC00356=527043
BC00357=519335
BC00358=519335
BC00359=550079
BC00360=550079
BC00361=542403
BC00362=542207
BC00363=506510
BC00364=542207
BC00365=519224
BC00366=542207
BC00367=492150
BC00368=423885
BC00369=471005
BC00370=487965
BC00371=477405
BC00372=472948
BC00373=455020
BC00374=453643
BC00375=453643
BC00376=493160
BC00377=521199
BC00378=521199
BC00379=521199
BC00380=521199
BC00381=484684
BC00382=484684
BC00383=484684
BC00384=484684
BC00385=484684
BC00386=484684
BC00387=484684
BC00388=493160
BC00389=582810
BC00390=655182
BC00391=655182
BC00392=655182
BC00393=655182
BC00394=716328
BC00395=716642
BC00396=582810
BC00397=493160
BC00398=542207
BC00399=542207
BC00400=505858
BC00401=590944
BC00402=557139
BC00403=543764
BC00404=551223
BC00405=543862
BC00406=551454
BC00407=589824
BC00408=589880
BC00409=589882
BC00410=589824
BC00411=600584
BC00412=608254
BC00413=600725
BC00414=600584
BC00415=588848
BC00416=532845
BC00417=543402
BC00418=533724
BC00419=584417
BC00420=590475
BC00421=610524
BC00422=594969
BC00423=594969
BC00424=594969
BC00425=593583
BC00426=552811
BC00427=552811
BC00428=552811
BC00429=552811
BC00430=612529
BC00431=612529
BC00432=620193
BC00433=620193
BC00434=620193
BC00435=620193
BC00436=620193
BC00437=620193
BC00438=620193
BC00439=812803
BC00440=887783
BC00441=897274
BC00442=900756
BC00443=946669
BC00444=910776
BC00445=910776
BC00446=924220
BC00447=853059
BC00448=542207
BC00449=542207
BC00450=542207
BC00451=542207
BC00452=574221
BC00453=593265
BC00454=574567
BC00455=599648
BC00456=600697
BC00457=605883
BC00458=605883
BC00459=605883
BC00460=617798
BC00461=617798
BC00462=617798
BC00463=666372
BC00464=666372
BC00465=725342
BC00466=740703
BC00467=740703
BC00468=740703
BC00469=710007
BC00470=710007
BC00471=703771
BC00472=710137
BC00473=710007
BC00474=727159
BC00475=725395
BC00476=733039
BC00477=733103
BC00478=733103
BC00479=733103
BC00480=733103
BC00481=733103
BC00482=733103
BC00483=733103
BC00484=620193
BC00485=626283
BC00486=635598
BC00487=635765
BC00488=635816
BC00489=643271
BC00490=641590
BC00491=641590
BC00492=685792
BC00493=685797
BC00494=685792
BC00495=685792
BC00496=685792
BC00497=771083
BC00498=750783
BC00499=758455
BC00500=750783
BC00501=750783
BC00502=719658
BC00503=685920
BC00504=620193
BC00505=620193
BC00506=561542
BC00507=498768
BC00508=407896
BC00509=407892
BC00510=469047
BC00511=469397
BC00512=524165
BC00513=524165
BC00514=733103
BC00515=733103
BC00516=733103
BC00517=733103
BC00518=733103
BC00519=733103
BC00520=771424
BC00521=771424
BC00522=779179
BC00523=771424
BC00524=794504
BC00525=794504
BC00526=801218
BC00527=794504
BC00528=840598
BC00529=840598
BC00530=846974
BC00531=840598
BC00532=840598
BC00533=840598
BC00534=840598
BC00535=840598
BC00536=795297
BC00537=741582
BC00538=733102
BC00539=620193
BC00540=700154
BC00541=704277
BC00542=716233
BC00543=716233
BC00544=716233
BC00545=716233
BC00546=716233
BC00547=733710
BC00548=733710
BC00549=733710
BC00550=733710
BC00551=742336
BC00552=742336
BC00553=742336
BC00554=763798
BC00555=742336
BC00556=742336
BC00557=742336
BC00558=742336
BC00559=743633
BC00560=750104
BC00561=672725
BC00562=672725
BC00563=672725
BC00564=576077
BC00565=465158
BC00566=407896
BC00567=407896
BC00568=407896
BC00569=407896
BC00570=407896
BC00571=407896
BC00572=471446
BC00573=524165
BC00574=524165
BC00575=733103
BC00576=733103
BC00577=733103
BC00578=733103
BC00579=733103
BC00580=733103
BC00581=830659
BC00582=830659
BC00583=837906
BC00584=830659
BC00585=825891
BC00586=830659
BC00587=830659
BC00588=828792
BC00589=818001
BC00590=822546
BC00591=814064
BC00592=794515
BC00593=795297
BC00594=733103
BC00595=733103
BC00596=762701
BC00597=816902
BC00598=816902
BC00599=837114
BC00600=816902
BC00601=816839
BC00602=816869
BC00603=816900
BC00604=816902
BC00605=816839
BC00606=816902
BC00607=837114
BC00608=903552
BC00609=903552
BC00610=897057
BC00611=903398
BC00612=903552
BC00613=903552
BC00614=903552
BC00615=903552
BC00616=903552
BC00617=903552
BC00618=903552
BC00619=848113
BC00620=815298
BC00621=672725
BC00622=672725
BC00623=672725
BC00624=576077
BC00625=513681
BC00626=534857
BC00627=557970
BC00628=557452
BC00629=618309
BC00630=618402
BC00631=618402
BC00632=618402
BC00633=618402
BC00634=733103
BC00635=733103
BC00636=931156
BC00637=923671
BC00638=923671
BC00639=923671
BC00640=947035
BC00641=947037
BC00642=947037
BC00643=954731
BC00644=953698
BC00645=953698
BC00646=953698
BC00647=953698
BC00648=953696
BC00649=953696
BC00650=953696
BC00651=927238
BC00652=910278
BC00653=910278
BC00654=917826
BC00655=907380
BC00656=917826
BC00657=914957
BC00658=898435
BC00659=840598
BC00660=795297
BC00661=748875
BC00662=852584
BC00663=921533
BC00664=921533
BC00665=923427
BC00666=923499
BC00667=923499
BC00668=923501
BC00669=932594
BC00670=943380
BC00671=943380
BC00672=943380
BC00673=963295
BC00674=934184
BC00675=929661
BC00676=754884
BC00677=672725
BC00678=672725
BC00679=749842
BC00680=756681
BC00681=776639
BC00682=776639
BC00683=776639
BC00684=838373
BC00685=837995
BC00686=796760
BC00687=742282
///POSTYPE BASE
///RECTAN
///RCONF 1,0,0,0,0,0,0,0,0,0,0,0,0,0,0,0,0,0,0,0,0,0,0,0
P00006=0.000,0.000,0.000,0.0000,0.0000,0.0000
///RCONF 0,0,0,0,0,0,0,0,0,0,0,0,0,0,0,0,0,0,0,0,0,0,0,0
P00058=0.000,0.000,3.000,0.0000,0.0000,0.0000
///RCONF 1,0,0,0,0,0,0,0,0,0,0,0,0,0,0,0,0,0,0,0,0,0,0,0
P00300=-0.036,-1.505,2.318,0.0000,0.0000,0.0000
P00301=0.046,-2.112,7.779,0.0000,0.0000,0.0000
P00302=-0.180,-2.409,6.326,0.0000,0.0000,0.0000
///RCONF 0,0,0,0,0,0,0,0,0,0,0,0,0,0,0,0,0,0,0,0,0,0,0,0
P00303=-0.004,-1.437,-4.584,0.0000,0.0000,0.0000
P00304=0.028,-1.666,-4.234,0.0000,0.0000,0.0000
P00305=-0.003,-1.920,-3.501,0.0000,0.0000,0.0000
P00306=0.015,-2.252,-3.054,0.0000,0.0000,0.0000
P00307=0.019,-2.151,-5.077,0.0000,0.0000,0.0000
P00308=-0.003,-2.092,-4.888,0.0000,0.0000,0.0000
P00309=-0.040,-2.205,-4.992,0.0000,0.0000,0.0000
P00310=-0.006,-2.490,-5.925,0.0000,0.0000,0.0000
P00311=-0.007,-2.079,-5.307,0.0000,0.0000,0.0000
P00312=-0.032,2.202,-7.632,0.0000,0.0000,0.0000
///RCONF 1,0,0,0,0,0,0,0,0,0,0,0,0,0,0,0,0,0,0,0,0,0,0,0
P00313=-0.088,1.055,2.110,0.0000,0.0000,0.0000
P00314=-0.055,1.752,1.634,0.0000,0.0000,0.0000
P00316=0.009,2.112,2.075,0.0000,0.0000,0.0000
P00317=-0.015,2.781,3.126,0.0000,0.0000,0.0000
P00318=-0.086,2.132,2.037,0.0000,0.0000,0.0000
///RCONF 0,0,0,0,0,0,0,0,0,0,0,0,0,0,0,0,0,0,0,0,0,0,0,0
P00350=11.519,-0.008,1.149,0.0000,0.0000,0.0000
P00351=13.563,-0.027,-0.653,0.0000,0.0000,0.0000
P00352=13.252,-0.027,-0.827,0.0000,0.0000,0.0000
P00353=10.971,-0.082,0.776,0.0000,0.0000,0.0000
P00354=-0.024,2.508,-1.824,0.0000,0.0000,0.0000
P00355=-0.001,2.528,-1.131,0.0000,0.0000,0.0000
P00356=-0.034,2.921,-0.262,0.0000,0.0000,0.0000
P00357=0.003,3.386,-0.091,0.0000,0.0000,0.0000
P00358=0.014,3.037,-0.020,0.0000,0.0000,0.0000
P00359=-0.005,2.731,0.912,0.0000,0.0000,0.0000
P00360=-0.011,3.412,0.438,0.0000,0.0000,0.0000
P00361=0.018,3.050,1.253,0.0000,0.0000,0.0000
P00401=3.430,-0.021,1.131,0.0000,0.0000,0.0000
P00402=-0.253,1.107,3.062,0.0000,0.0000,0.0000
P00403=-3.666,-0.015,5.328,0.0000,0.0000,0.0000
///RCONF 1,0,0,0,0,0,0,0,0,0,0,0,0,0,0,0,0,0,0,0,0,0,0,0
P00404=0.029,4.189,-1.030,0.0000,0.0000,0.0000
///RCONF 0,0,0,0,0,0,0,0,0,0,0,0,0,0,0,0,0,0,0,0,0,0,0,0
P00405=2.420,0.007,1.427,0.0000,0.0000,0.0000
P00406=3.513,-0.022,0.429,0.0000,0.0000,0.0000
///RCONF 1,0,0,0,1,0,0,0,0,0,0,0,0,0,0,0,0,0,0,0,0,0,0,0
P00407=-0.029,2.348,-1.469,0.0000,0.0000,0.0000
P00408=0.010,1.346,-1.479,0.0000,0.0000,0.0000
///RCONF 1,0,0,0,0,0,0,0,0,0,0,0,0,0,0,0,0,0,0,0,0,0,0,0
P00409=-0.026,2.090,-1.483,0.0000,0.0000,0.0000
P00410=0.001,4.491,-0.583,0.0000,0.0000,0.0000
///RCONF 1,0,0,0,1,0,0,0,0,0,0,0,0,0,0,0,0,0,0,0,0,0,0,0
P00411=-0.015,3.627,0.872,0.0000,0.0000,0.0000
P00412=0.002,3.829,0.787,0.0000,0.0000,0.0000
P00413=0.046,0.107,-0.040,0.0000,0.0000,0.0000
///RCONF 1,0,0,0,0,0,0,0,0,0,0,0,0,0,0,0,0,0,0,0,0,0,0,0
P00414=0.046,0.800,0.739,0.0000,0.0000,0.0000
///RCONF 0,0,0,0,0,0,0,0,0,0,0,0,0,0,0,0,0,0,0,0,0,0,0,0
P00415=-1.781,-1.303,3.250,0.0000,0.0000,0.0000
P00416=0.027,1.119,3.078,0.0000,0.0000,0.0000
///RCONF 1,0,0,0,1,0,0,0,0,0,0,0,0,0,0,0,0,0,0,0,0,0,0,0
P00417=0.059,4.721,3.973,0.0000,0.0000,0.0000
//INST
///DATE 2024/07/04 14:18
///ATTR SC,RW
///GROUP1 RB1,BS1
NOP
CALL JOB:MOVE_INTO_TUNNEL
MOVJ C00000 BC00000 VJ=50.00
MOVJ C00001 BC00001 VJ=40.00
MOVJ C00002 BC00002 VJ=40.00
MOVL C00003 BC00003 V=666.7
MOVJ C00004 BC00004 VJ=30.00
MOVL C00005 BC00005 V=500.0
'------------------------
'W31.2
'------------------------
MOVL C00006 BC00006 V=166.7 PL=0
REFP 3 C00007 BC00007
CALL JOB:SEARCH-R1
SET P0300 P0006
SFTON P0300
MOVL C00008 BC00008 V=166.7 PL=0
REFP 3 C00009 BC00009
CALL JOB:SEARCH-R1
SET P0300 P0006
SFTON P0300
MOVL C00010 BC00010 V=166.7 PL=0
SFTOF
'------------------------
'W31.4
'------------------------
MOVL C00011 BC00011 V=500.0
MOVL C00012 BC00012 V=166.7 PL=0
REFP 3 C00013 BC00013
CALL JOB:SEARCH-R1
SET P0301 P0006
SFTON P0301
MOVL C00014 BC00014 V=166.7 PL=0
REFP 3 C00015 BC00015
CALL JOB:SEARCH-R1
SET P0301 P0006
SFTON P0301
MOVL C00016 BC00016 V=166.7 PL=0
SFTOF
'------------------------
'W31.6
'------------------------
MOVL C00017 BC00017 V=500.0
MOVL C00018 BC00018 V=166.7 PL=0
REFP 3 C00019 BC00019
CALL JOB:SEARCH-R1
SET P0302 P0006
SFTON P0302
MOVL C00020 BC00020 V=166.7 PL=0
REFP 3 C00021 BC00021
CALL JOB:SEARCH-R1
SET P0302 P0006
SFTON P0302
MOVL C00022 BC00022 V=166.7 PL=0
SFTOF
'------------------------
'W31.8
'------------------------
MOVL C00023 BC00023 V=500.0
MOVL C00024 BC00024 V=166.7 PL=0
REFP 3 C00025 BC00025
CALL JOB:SEARCH-R1
SET P0303 P0006
SFTON P0303
MOVL C00026 BC00026 V=166.7 PL=0
REFP 3 C00027 BC00027
CALL JOB:SEARCH-R1
SET P0303 P0006
SFTON P0303
MOVL C00028 BC00028 V=166.7 PL=0
SFTOF
'------------------------
'W31.9
'------------------------
MOVL C00029 BC00029 V=500.0
MOVL C00030 BC00030 V=166.7 PL=0
REFP 3 C00031 BC00031
CALL JOB:SEARCH-R1
SET P0304 P0006
SFTON P0304
MOVL C00032 BC00032 V=166.7 PL=0
REFP 3 C00033 BC00033
CALL JOB:SEARCH-R1
SET P0304 P0006
SFTON P0304
MOVL C00034 BC00034 V=166.7 PL=0
SFTOF
'------------------------
'W31.11
'------------------------
MOVL C00035 BC00035 V=500.0
MOVL C00036 BC00036 V=166.7 PL=0
REFP 3 C00037 BC00037
CALL JOB:SEARCH-R1
SET P0305 P0006
SFTON P0305
MOVL C00038 BC00038 V=166.7 PL=0
REFP 3 C00039 BC00039
CALL JOB:SEARCH-R1
SET P0305 P0006
SFTON P0305
MOVL C00040 BC00040 V=166.7 PL=0
SFTOF
'------------------------
'W31.13
'------------------------
MOVL C00041 BC00041 V=500.0
MOVL C00042 BC00042 V=166.7 PL=0
REFP 3 C00043 BC00043
CALL JOB:SEARCH-R1
SET P0306 P0006
SFTON P0306
MOVL C00044 BC00044 V=166.7 PL=0
REFP 3 C00045 BC00045
CALL JOB:SEARCH-R1
SET P0306 P0006
SFTON P0306
MOVL C00046 BC00046 V=166.7 PL=0
SFTOF
'------------------------
'W31.14
'------------------------
MOVL C00047 BC00047 V=500.0
MOVL C00048 BC00048 V=166.7 PL=0
REFP 3 C00049 BC00049
CALL JOB:SEARCH-R1
SET P0307 P0006
SFTON P0307
MOVL C00050 BC00050 V=166.7 PL=0
REFP 3 C00051 BC00051
CALL JOB:SEARCH-R1
SET P0307 P0006
SFTON P0307
MOVL C00052 BC00052 V=166.7 PL=0
SFTOF
'------------------------
'W31.16
'------------------------
MOVL C00053 BC00053 V=500.0
MOVL C00054 BC00054 V=166.7 PL=0
REFP 3 C00055 BC00055
CALL JOB:SEARCH-R1
SET P0308 P0006
SFTON P0308
MOVL C00056 BC00056 V=166.7 PL=0
REFP 3 C00057 BC00057
CALL JOB:SEARCH-R1
SET P0308 P0006
SFTON P0308
MOVL C00058 BC00058 V=166.7 PL=0
SFTOF
MOVL C00059 BC00059 V=150.0
MOVL C00060 BC00060 V=333.3
MOVL C00061 BC00061 V=500.0
MOVL C00062 BC00062 V=500.0
MOVJ C00063 BC00063 VJ=50.00
MOVL C00064 BC00064 V=666.7
MOVL C00065 BC00065 V=500.0
MOVL C00066 BC00066 V=333.3
'------------------------
'W31.18
'------------------------
MOVL C00067 BC00067 V=166.7
MOVL C00068 BC00068 V=133.3 PL=0
REFP 3 C00069 BC00069
CALL JOB:SEARCH-R1
SET P0309 P0006
SFTON P0309
MOVL C00070 BC00070 V=66.7 PL=0
REFP 3 C00071 BC00071
CALL JOB:SEARCH-R1
SET P0309 P0006
SFTON P0309
MOVL C00072 BC00072 V=66.7 PL=0
SFTOF
'------------------------
'W31.19
'------------------------
MOVL C00073 BC00073 V=500.0
MOVL C00074 BC00074 V=166.7 PL=0
REFP 3 C00075 BC00075
CALL JOB:SEARCH-R1
SET P0310 P0006
SFTON P0310
MOVL C00076 BC00076 V=166.7 PL=0
REFP 3 C00077 BC00077
CALL JOB:SEARCH-R1
SET P0310 P0006
SFTON P0310
MOVL C00078 BC00078 V=166.7 PL=0
SFTOF
'------------------------
'W31.21
'------------------------
MOVL C00079 BC00079 V=500.0
MOVL C00080 BC00080 V=166.7 PL=0
REFP 3 C00081 BC00081
CALL JOB:SEARCH-R1
SET P0311 P0006
SFTON P0311
MOVL C00082 BC00082 V=166.7 PL=0
REFP 3 C00083 BC00083
CALL JOB:SEARCH-R1
SET P0311 P0006
SFTON P0311
MOVL C00084 BC00084 V=166.7 PL=0
SFTOF
'------------------------
'W31.22
'------------------------
MOVL C00085 BC00085 V=500.0
MOVL C00086 BC00086 V=166.7 PL=0
REFP 3 C00087 BC00087
CALL JOB:SEARCH-R1
SET P0312 P0006
SFTON P0312
MOVL C00088 BC00088 V=166.7 PL=0
REFP 3 C00089 BC00089
CALL JOB:SEARCH-R1
SET P0312 P0006
SFTON P0312
MOVL C00090 BC00090 V=166.7 PL=0
SFTOF
'------------------------
'W31.24
'------------------------
MOVL C00091 BC00091 V=500.0
MOVL C00092 BC00092 V=166.7 PL=0
REFP 3 C00093 BC00093
CALL JOB:SEARCH-R1
SET P0313 P0006
SFTON P0313
MOVL C00094 BC00094 V=166.7 PL=0
REFP 3 C00095 BC00095
CALL JOB:SEARCH-R1
SET P0313 P0006
SFTON P0313
MOVL C00096 BC00096 V=166.7 PL=0
SFTOF
'------------------------
'W31.26
'------------------------
MOVL C00097 BC00097 V=500.0
MOVL C00098 BC00098 V=166.7 PL=0
REFP 3 C00099 BC00099
CALL JOB:SEARCH-R1
SET P0314 P0006
SFTON P0314
MOVL C00100 BC00100 V=166.7 PL=0
REFP 3 C00101 BC00101
CALL JOB:SEARCH-R1
SET P0314 P0006
SFTON P0314
MOVL C00102 BC00102 V=166.7 PL=0
SFTOF
'------------------------
MOVL C00103 BC00103 V=333.3
MOVL C00104 BC00104 V=666.7
MOVL C00105 BC00105 V=666.7
MOVL C00106 BC00106 V=666.7
MOVL C00107 BC00107 V=666.7
MOVL C00108 BC00108 V=666.7
MOVL C00109 BC00109 V=666.7
MOVL C00110 BC00110 V=333.3
MOVL C00111 BC00111 V=250.0
'------------------------
'W31.29
'------------------------
MOVL C00112 BC00112 V=166.7 PL=0
REFP 3 C00113 BC00113
CALL JOB:SEARCH-R1
SET P0316 P0006
SFTON P0316
MOVL C00114 BC00114 V=166.7 PL=0
REFP 3 C00115 BC00115
CALL JOB:SEARCH-R1
SET P0316 P0006
SFTON P0316
MOVL C00116 BC00116 V=166.7 PL=0
SFTOF
'------------------------
'W31.31
'------------------------
MOVL C00117 BC00117 V=500.0
MOVL C00118 BC00118 V=166.7 PL=0
REFP 3 C00119 BC00119
CALL JOB:SEARCH-R1
SET P0317 P0006
SFTON P0317
MOVL C00120 BC00120 V=166.7 PL=0
REFP 3 C00121 BC00121
CALL JOB:SEARCH-R1
SET P0317 P0006
SFTON P0317
MOVL C00122 BC00122 V=166.7 PL=0
SFTOF
'------------------------
'W31.32
'------------------------
MOVL C00123 BC00123 V=250.0
MOVL C00124 BC00124 V=166.7 PL=0
REFP 3 C00125 BC00125
CALL JOB:SEARCH-R1
SET P0318 P0006
SFTON P0318
MOVL C00126 BC00126 V=166.7 PL=0
REFP 3 C00127 BC00127
CALL JOB:SEARCH-R1
SET P0318 P0006
SFTON P0318
MOVL C00128 BC00128 V=166.7 PL=0
SFTOF
MOVL C00129 BC00129 V=250.0
MOVL C00130 BC00130 V=333.3
MOVL C00131 BC00131 V=333.3
MOVL C00132 BC00132 V=666.7
MOVJ C00133 BC00133 VJ=50.00
MOVJ C00134 BC00134 VJ=50.00
MOVJ C00135 BC00135 VJ=50.00
MOVJ C00136 BC00136 VJ=50.00
MOVJ C00137 BC00137 VJ=30.00
MOVL C00138 BC00138 V=166.7
'------------------------
'W214B L
'------------------------
MOVL C00139 BC00139 V=166.7 PL=0
REFP 3 C00140 BC00140
CALL JOB:SEARCH-R1
IMOV P0058 V=16.7
SET P0350 P0006
SFTON P0350
REFP 3 C00141 BC00141
CALL JOB:SEARCH-R1
SET P0350 P0006
SFTON P0350
MOVL C00142 BC00142 V=166.7 PL=0
SFTOF
'------------------------
'W214A P
'------------------------
MOVJ C00143 BC00143 VJ=40.00
MOVL C00144 BC00144 V=166.7 PL=0
REFP 3 C00145 BC00145
CALL JOB:SEARCH-R1
IMOV P0058 V=16.7
SET P0351 P0006
SFTON P0351
REFP 3 C00146 BC00146
CALL JOB:SEARCH-R1
SET P0351 P0006
SFTON P0351
MOVL C00147 BC00147 V=166.7 PL=0
SFTOF
'------------------------
'W219B L
'------------------------
MOVJ C00148 BC00148 VJ=40.00
MOVL C00149 BC00149 V=166.7 PL=0
REFP 3 C00150 BC00150
CALL JOB:SEARCH-R1
IMOV P0058 V=16.7
SET P0352 P0006
SFTON P0352
REFP 3 C00151 BC00151
CALL JOB:SEARCH-R1
SET P0352 P0006
SFTON P0352
MOVL C00152 BC00152 V=166.7 PL=0
SFTOF
'------------------------
'W219B P
'------------------------
MOVJ C00153 BC00153 VJ=40.00
MOVL C00154 BC00154 V=166.7 PL=0
REFP 3 C00155 BC00155
CALL JOB:SEARCH-R1
IMOV P0058 V=16.7
SET P0353 P0006
SFTON P0353
REFP 3 C00156 BC00156
CALL JOB:SEARCH-R1
SET P0353 P0006
SFTON P0353
MOVL C00157 BC00157 V=166.7 PL=0
SFTOF
'------------------------
'W213B L
'------------------------
MOVJ C00158 BC00158 VJ=40.00
MOVL C00159 BC00159 V=166.7 PL=0
REFP 3 C00160 BC00160
CALL JOB:SEARCH-R1
IMOV P0058 V=16.7
SET P0354 P0006
SFTON P0354
REFP 3 C00161 BC00161
CALL JOB:SEARCH-R1
SET P0354 P0006
SFTON P0354
MOVL C00162 BC00162 V=166.7 PL=0
SFTOF
'------------------------
'W213B P
'------------------------
MOVJ C00163 BC00163 VJ=40.00
MOVL C00164 BC00164 V=166.7 PL=0
REFP 3 C00165 BC00165
CALL JOB:SEARCH-R1
IMOV P0058 V=16.7
SET P0355 P0006
SFTON P0355
REFP 3 C00166 BC00166
CALL JOB:SEARCH-R1
SET P0355 P0006
SFTON P0355
MOVL C00167 BC00167 V=166.7 PL=0
SFTOF
'------------------------
'W218B L
'------------------------
MOVJ C00168 BC00168 VJ=40.00
MOVL C00169 BC00169 V=166.7 PL=0
REFP 3 C00170 BC00170
CALL JOB:SEARCH-R1
IMOV P0058 V=16.7
SET P0356 P0006
SFTON P0356
REFP 3 C00171 BC00171
CALL JOB:SEARCH-R1
SET P0356 P0006
SFTON P0356
MOVL C00172 BC00172 V=166.7 PL=0
SFTOF
'------------------------
'W218B P
'------------------------
MOVJ C00173 BC00173 VJ=40.00
MOVL C00174 BC00174 V=166.7 PL=0
REFP 3 C00175 BC00175
CALL JOB:SEARCH-R1
IMOV P0058 V=16.7
SET P0357 P0006
SFTON P0357
REFP 3 C00176 BC00176
CALL JOB:SEARCH-R1
SET P0357 P0006
SFTON P0357
MOVL C00177 BC00177 V=166.7 PL=0
SFTOF
'------------------------
'W215B L
'------------------------
MOVJ C00178 BC00178 VJ=40.00
MOVL C00179 BC00179 V=166.7 PL=0
REFP 3 C00180 BC00180
CALL JOB:SEARCH-R1
IMOV P0058 V=16.7
SET P0358 P0006
SFTON P0358
REFP 3 C00181 BC00181
CALL JOB:SEARCH-R1
SET P0358 P0006
SFTON P0358
MOVL C00182 BC00182 V=166.7 PL=0
SFTOF
'------------------------
'W215B P
'------------------------
MOVL C00183 BC00183 V=666.7
MOVL C00184 BC00184 V=166.7 PL=0
REFP 3 C00185 BC00185
CALL JOB:SEARCH-R1
IMOV P0058 V=16.7
SET P0359 P0006
SFTON P0359
REFP 3 C00186 BC00186
CALL JOB:SEARCH-R1
SET P0359 P0006
SFTON P0359
MOVL C00187 BC00187 V=166.7 PL=0
SFTOF
'------------------------
'W217B L
'------------------------
MOVL C00188 BC00188 V=666.7
MOVL C00189 BC00189 V=166.7 PL=0
REFP 3 C00190 BC00190
CALL JOB:SEARCH-R1
IMOV P0058 V=16.7
SET P0360 P0006
SFTON P0360
REFP 3 C00191 BC00191
CALL JOB:SEARCH-R1
SET P0360 P0006
SFTON P0360
MOVL C00192 BC00192 V=166.7 PL=0
SFTOF
'------------------------
'W217B P
'------------------------
MOVL C00193 BC00193 V=666.7
MOVL C00194 BC00194 V=166.7 PL=0
REFP 3 C00195 BC00195
CALL JOB:SEARCH-R1
IMOV P0058 V=16.7
SET P0361 P0006
SFTON P0361
REFP 3 C00196 BC00196
CALL JOB:SEARCH-R1
SET P0361 P0006
SFTON P0361
MOVL C00197 BC00197 V=166.7 PL=0
SFTOF
MOVL C00198 BC00198 V=333.3
MOVL C00199 BC00199 V=666.7
MOVL C00200 BC00200 V=666.7
MOVJ C00201 BC00201 VJ=50.00
MOVJ C00202 BC00202 VJ=50.00
COMM MOVJ C00203 BC00203 VJ=40.00
COMM MOVJ C00204 BC00204 VJ=40.00
COMM MOVJ C00205 BC00205 VJ=25.00
COMM MOVJ C00206 BC00206 VJ=30.00
COMM MOVJ C00207 BC00207 VJ=30.00
COMM MOVJ C00208 BC00208 VJ=20.00
COMM MOVL C00209 BC00209 V=500.0
COMM '------------------------
COMM 'W27.4
COMM '------------------------
COMM MOVL C00210 BC00210 V=166.7 PL=0
COMM REFP 3 C00211 BC00211
COMM CALL JOB:SEARCH-R1
COMM SET P0401 P0006
COMM SFTON P0401
COMM MOVL C00212 BC00212 V=166.7 PL=0
COMM REFP 3 C00213 BC00213
COMM CALL JOB:SEARCH-R1
COMM SET P0401 P0006
COMM SFTON P0401
COMM MOVL C00214 BC00214 V=166.7 PL=0
COMM SFTOF
COMM '------------------------
COMM 'W27.6
COMM '------------------------
COMM MOVL C00215 BC00215 V=666.7
COMM MOVL C00216 BC00216 V=166.7 PL=0
COMM REFP 3 C00217 BC00217
COMM CALL JOB:SEARCH-R1
COMM SET P0402 P0006
COMM SFTON P0402
COMM MOVL C00218 BC00218 V=166.7 PL=0
COMM REFP 3 C00219 BC00219
COMM CALL JOB:SEARCH-R1
COMM SET P0402 P0006
COMM SFTON P0402
COMM MOVL C00220 BC00220 V=166.7 PL=0
COMM SFTOF
COMM MOVL C00221 BC00221 V=500.0
COMM MOVL C00222 BC00222 V=500.0
COMM '------------------------
COMM 'W27.8
COMM '------------------------
COMM MOVL C00223 BC00223 V=333.3
COMM MOVL C00224 BC00224 V=166.7 PL=0
COMM REFP 3 C00225 BC00225
COMM CALL JOB:SEARCH-R1
COMM SET P0403 P0006
COMM SFTON P0403
COMM MOVL C00226 BC00226 V=166.7 PL=0
COMM REFP 3 C00227 BC00227
COMM CALL JOB:SEARCH-R1
COMM SET P0403 P0006
COMM SFTON P0403
COMM MOVL C00228 BC00228 V=166.7 PL=0
COMM SFTOF
COMM MOVJ C00229 BC00229 VJ=25.00
COMM MOVJ C00230 BC00230 VJ=25.00
COMM MOVJ C00231 BC00231 VJ=30.00
COMM MOVJ C00232 BC00232 VJ=40.00
COMM MOVJ C00233 BC00233 VJ=30.00
COMM '------------------------
COMM 'W27.9
COMM '------------------------
COMM MOVL C00234 BC00234 V=500.0
COMM MOVL C00235 BC00235 V=166.7 PL=0
COMM REFP 3 C00236 BC00236
COMM CALL JOB:SEARCH-R1
COMM SET P0404 P0006
COMM SFTON P0404
COMM MOVL C00237 BC00237 V=166.7 PL=0
COMM REFP 3 C00238 BC00238
COMM CALL JOB:SEARCH-R1
COMM SET P0404 P0006
COMM SFTON P0404
COMM MOVL C00239 BC00239 V=166.7 PL=0
COMM SFTOF
COMM MOVL C00240 BC00240 V=500.0
COMM '------------------------
COMM 'W27.11
COMM '------------------------
COMM MOVL C00241 BC00241 V=500.0
COMM MOVL C00242 BC00242 V=166.7 PL=0
COMM REFP 3 C00243 BC00243
COMM CALL JOB:SEARCH-R1
COMM SET P0405 P0006
COMM SFTON P0405
COMM MOVL C00244 BC00244 V=166.7 PL=0
COMM REFP 3 C00245 BC00245
COMM CALL JOB:SEARCH-R1
COMM SET P0405 P0006
COMM SFTON P0405
COMM MOVL C00246 BC00246 V=166.7 PL=0
COMM SFTOF
COMM MOVL C00247 BC00247 V=666.7
COMM MOVL C00248 BC00248 V=666.7
COMM '------------------------
COMM 'W27.13
COMM '------------------------
COMM MOVL C00249 BC00249 V=333.3
COMM MOVL C00250 BC00250 V=166.7 PL=0
COMM REFP 3 C00251 BC00251
COMM CALL JOB:SEARCH-R1
COMM SET P0406 P0006
COMM SFTON P0406
COMM MOVL C00252 BC00252 V=166.7 PL=0
COMM REFP 3 C00253 BC00253
COMM CALL JOB:SEARCH-R1
COMM SET P0406 P0006
COMM SFTON P0406
COMM MOVL C00254 BC00254 V=166.7 PL=0
COMM SFTOF
COMM '------------------------
COMM 'W27.14
COMM '------------------------
COMM MOVL C00255 BC00255 V=666.7
COMM MOVL C00256 BC00256 V=166.7 PL=0
COMM REFP 3 C00257 BC00257
COMM CALL JOB:SEARCH-R1
COMM SET P0407 P0006
COMM SFTON P0407
COMM MOVL C00258 BC00258 V=166.7 PL=0
COMM REFP 3 C00259 BC00259
COMM CALL JOB:SEARCH-R1
COMM SET P0407 P0006
COMM SFTON P0407
COMM MOVL C00260 BC00260 V=166.7 PL=0
COMM SFTOF
COMM MOVL C00261 BC00261 V=666.7
COMM '------------------------
COMM 'W27.16
COMM '------------------------
COMM MOVL C00262 BC00262 V=333.3
COMM MOVL C00263 BC00263 V=166.7 PL=0
COMM REFP 3 C00264 BC00264
COMM CALL JOB:SEARCH-R1
COMM SET P0408 P0006
COMM SFTON P0408
COMM MOVL C00265 BC00265 V=166.7 PL=0
COMM REFP 3 C00266 BC00266
COMM CALL JOB:SEARCH-R1
COMM SET P0408 P0006
COMM SFTON P0408
COMM MOVL C00267 BC00267 V=166.7 PL=0
COMM SFTOF
COMM MOVL C00268 BC00268 V=666.7
COMM MOVJ C00269 BC00269 VJ=30.00
COMM MOVJ C00270 BC00270 VJ=50.00
COMM MOVJ C00271 BC00271 VJ=40.00
COMM MOVJ C00272 BC00272 VJ=30.00
COMM '------------------------
COMM 'W27.18
COMM '------------------------
COMM MOVL C00273 BC00273 V=333.3
COMM MOVL C00274 BC00274 V=166.7 PL=0
COMM REFP 3 C00275 BC00275
COMM CALL JOB:SEARCH-R1
COMM SET P0409 P0006
COMM SFTON P0409
COMM MOVL C00276 BC00276 V=166.7 PL=0
COMM REFP 3 C00277 BC00277
COMM CALL JOB:SEARCH-R1
COMM SET P0409 P0006
COMM SFTON P0409
COMM MOVL C00278 BC00278 V=166.7 PL=0
COMM SFTOF
COMM '------------------------
COMM 'W27.19
COMM '------------------------
COMM MOVL C00279 BC00279 V=666.7
COMM MOVL C00280 BC00280 V=166.7 PL=0
COMM REFP 3 C00281 BC00281
COMM CALL JOB:SEARCH-R1
COMM SET P0410 P0006
COMM SFTON P0410
COMM MOVL C00282 BC00282 V=166.7 PL=0
COMM REFP 3 C00283 BC00283
COMM CALL JOB:SEARCH-R1
COMM SET P0410 P0006
COMM SFTON P0410
COMM MOVL C00284 BC00284 V=166.7 PL=0
COMM SFTOF
COMM MOVL C00285 BC00285 V=666.7
COMM '------------------------
COMM 'W27.21
COMM '------------------------
COMM MOVL C00286 BC00286 V=166.7 PL=0
COMM REFP 3 C00287 BC00287
COMM CALL JOB:SEARCH-R1
COMM SET P0411 P0006
COMM SFTON P0411
COMM MOVL C00288 BC00288 V=166.7 PL=0
COMM REFP 3 C00289 BC00289
COMM CALL JOB:SEARCH-R1
COMM SET P0411 P0006
COMM SFTON P0411
COMM MOVL C00290 BC00290 V=166.7 PL=0
COMM SFTOF
COMM '------------------------
COMM 'W27.22
COMM '------------------------
COMM MOVL C00291 BC00291 V=666.7
COMM MOVL C00292 BC00292 V=166.7 PL=0
COMM REFP 3 C00293 BC00293
COMM CALL JOB:SEARCH-R1
COMM SET P0412 P0006
COMM SFTON P0412
COMM MOVL C00294 BC00294 V=166.7 PL=0
COMM REFP 3 C00295 BC00295
COMM CALL JOB:SEARCH-R1
COMM SET P0412 P0006
COMM SFTON P0412
COMM MOVL C00296 BC00296 V=166.7 PL=0
COMM SFTOF
COMM MOVL C00297 BC00297 V=666.7
COMM MOVJ C00298 BC00298 VJ=30.00
COMM MOVL C00299 BC00299 V=500.0
COMM '------------------------
COMM 'W27.24
COMM '------------------------
COMM MOVL C00300 BC00300 V=666.7
COMM MOVL C00301 BC00301 V=166.7 PL=0
COMM REFP 3 C00302 BC00302
COMM CALL JOB:SEARCH-R1
COMM SET P0413 P0006
COMM SFTON P0413
COMM MOVL C00303 BC00303 V=166.7 PL=0
COMM REFP 3 C00304 BC00304
COMM CALL JOB:SEARCH-R1
COMM SET P0413 P0006
COMM SFTON P0413
COMM MOVL C00305 BC00305 V=166.7 PL=0
COMM SFTOF
COMM MOVL C00306 BC00306 V=666.7
COMM MOVJ C00307 BC00307 VJ=50.00
COMM MOVJ C00308 BC00308 VJ=50.00
COMM MOVJ C00309 BC00309 VJ=50.00
COMM MOVJ C00310 BC00310 VJ=20.00
COMM MOVJ C00311 BC00311 VJ=10.00
COMM '------------------------
COMM 'W27.26
COMM '------------------------
COMM MOVL C00312 BC00312 V=333.3
COMM MOVL C00313 BC00313 V=166.7 PL=0
COMM REFP 3 C00314 BC00314
COMM CALL JOB:SEARCH-R1
COMM SET P0414 P0006
COMM SFTON P0414
COMM MOVL C00315 BC00315 V=166.7 PL=0
COMM REFP 3 C00316 BC00316
COMM CALL JOB:SEARCH-R1
COMM SET P0414 P0006
COMM SFTON P0414
COMM MOVL C00317 BC00317 V=166.7 PL=0
COMM SFTOF
COMM MOVL C00318 BC00318 V=333.3
COMM MOVJ C00319 BC00319 VJ=30.00
COMM MOVJ C00320 BC00320 VJ=30.00
COMM MOVJ C00321 BC00321 VJ=30.00
COMM GETE D040 P0414 (1)
COMM GETE D041 P0414 (2)
COMM GETE D042 P0414 (3)
COMM SETE P0415 (1) D040
COMM SETE P0415 (2) D041
COMM SETE P0415 (3) D042
COMM '------------------------
COMM 'W27.29
COMM '------------------------
COMM MOVJ C00322 BC00322 VJ=30.00
COMM MOVJ C00323 BC00323 VJ=30.00
COMM MOVL C00324 BC00324 V=333.3
COMM MOVL C00325 BC00325 V=166.7 PL=0
COMM REFP 3 C00326 BC00326
COMM CALL JOB:SEARCH-R1
COMM SET P0416 P0006
COMM SFTON P0416
COMM MOVL C00327 BC00327 V=166.7 PL=0
COMM REFP 3 C00328 BC00328
COMM CALL JOB:SEARCH-R1
COMM SET P0416 P0006
COMM SFTON P0416
COMM MOVL C00329 BC00329 V=166.7 PL=0
COMM SFTOF
COMM '------------------------
COMM 'W27.31
COMM '------------------------
COMM MOVL C00330 BC00330 V=666.7
COMM MOVL C00331 BC00331 V=166.7 PL=0
COMM REFP 3 C00332 BC00332
COMM CALL JOB:SEARCH-R1
COMM SET P0417 P0006
COMM SFTON P0417
COMM MOVL C00333 BC00333 V=166.7 PL=0
COMM REFP 3 C00334 BC00334
COMM CALL JOB:SEARCH-R1
COMM SET P0417 P0006
COMM SFTON P0417
COMM MOVL C00335 BC00335 V=166.7 PL=0
COMM SFTOF
COMM '------------------------
COMM 'W27.32
COMM '------------------------
COMM MOVL C00336 BC00336 V=333.3
MOVJ C00337 BC00337 VJ=50.00
CALL JOB:FRONT_SEARCH_-90ST-1_4840
MOVJ C00338 BC00338 VJ=50.00
MOVJ C00339 BC00339 VJ=50.00
MOVJ C00340 BC00340 VJ=50.00
MOVL C00341 BC00341 V=666.7
MOVJ C00342 BC00342 VJ=30.00
'------------------------
'W31.2
'------------------------
SFTON P0300
MOVL C00343 BC00343 V=333.3
MOVL C00344 BC00344 V=166.7 PL=0
MACRO1 MJ#(0) ARGF10
ARCON
MOVL C00345 BC00345 V=10.8
ARCOF
MOVL C00346 BC00346 V=166.7
SFTOF
'------------------------
'W31.4
'------------------------
SFTON P0301
MOVL C00347 BC00347 V=666.7
MOVL C00348 BC00348 V=166.7 PL=0
ARCON
MOVL C00349 BC00349 V=10.8
ARCOF
MOVL C00350 BC00350 V=166.7
SFTOF
'------------------------
'W31.6
'------------------------
SFTON P0302
MOVL C00351 BC00351 V=666.7
MOVL C00352 BC00352 V=166.7 PL=0
ARCON
MOVL C00353 BC00353 V=10.8
ARCOF
MOVL C00354 BC00354 V=166.7
SFTOF
'------------------------
'W31.8
'------------------------
SFTON P0303
MOVL C00355 BC00355 V=666.7
MOVL C00356 BC00356 V=166.7 PL=0
ARCON
MOVL C00357 BC00357 V=10.8
ARCOF
MOVL C00358 BC00358 V=166.7
SFTOF
'------------------------
'W31.9
'------------------------
SFTON P0304
MOVL C00359 BC00359 V=666.7
MOVL C00360 BC00360 V=166.7 PL=0
ARCON
MOVL C00361 BC00361 V=10.8
ARCOF
MOVL C00362 BC00362 V=166.7
SFTOF
MOVL C00363 BC00363 V=500.0
MOVL C00364 BC00364 V=500.0
MOVJ C00365 BC00365 VJ=50.00
MOVJ C00366 BC00366 VJ=50.00
COMM '::::::::::::::::::::::::::::::::
COMM '::::::::::::::::::::::::::::::::
COMM '::::::::::::::::::::::::::::::::
COMM '::::::::::::::::::::::::::::::::
COMM '::::::::::::::::::::::::::::::::
COMM MOVJ C00367 BC00367 VJ=40.00
COMM MOVJ C00368 BC00368 VJ=40.00
COMM MOVJ C00369 BC00369 VJ=40.00
COMM MOVJ C00370 BC00370 VJ=40.00
COMM MOVJ C00371 BC00371 VJ=40.00
COMM MOVJ C00372 BC00372 VJ=40.00
COMM '------------------------
COMM 'W27.2
COMM '------------------------
COMM MOVL C00373 BC00373 V=500.0
COMM SFTON P0401
COMM MOVL C00374 BC00374 V=166.7 PL=0
COMM MACRO1 MJ#(0) ARGF24
COMM ARCON
COMM MOVL C00375 BC00375 V=7.5
COMM ARCOF
COMM SFTOF
COMM 'BELKA PRZEJAZD
COMM MOVL C00376 BC00376 V=500.0
COMM '------------------------
COMM 'W27.6
COMM '------------------------
COMM SFTON P0402
COMM MOVL C00377 BC00377 V=500.0
COMM MOVL C00378 BC00378 V=166.7 PL=0
COMM MACRO1 MJ#(0) ARGF24
COMM ARCON
COMM MOVL C00379 BC00379 V=7.5
COMM ARCOF
COMM MOVL C00380 BC00380 V=166.7
COMM SFTOF
COMM MOVJ C00381 BC00381 VJ=20.00
COMM '------------------------
COMM 'W27.8
COMM '------------------------
COMM SFTON P0403
COMM MOVL C00382 BC00382 V=500.0
COMM MOVL C00383 BC00383 V=166.7 PL=0
COMM MACRO1 MJ#(0) ARGF24
COMM ARCON
COMM MOVL C00384 BC00384 V=7.5
COMM ARCOF
COMM MOVL C00385 BC00385 V=166.7
COMM SFTOF
COMM MOVL C00386 BC00386 V=500.0
COMM MOVJ C00387 BC00387 VJ=50.00
MOVJ C00388 BC00388 VJ=50.00
MOVJ C00389 BC00389 VJ=50.00
MOVJ C00390 BC00390 VJ=50.00
MOVL C00391 BC00391 V=666.7
'------------------------
'W213A
'------------------------
SFTON P0355
MOVL C00392 BC00392 V=666.7
MOVL C00393 BC00393 V=166.7 PL=0
MACRO1 MJ#(0) ARGF9
ARCON
SFTOF
SFTON P0354
MOVL C00394 BC00394 V=11.2
ARCOF
MOVL C00395 BC00395 V=333.3
SFTOF
MOVJ C00396 BC00396 VJ=50.00
MOVJ C00397 BC00397 VJ=50.00
MOVJ C00398 BC00398 VJ=50.00
MOVJ C00399 BC00399 VJ=50.00
MOVJ C00400 BC00400 VJ=30.00
MOVJ C00401 BC00401 VJ=20.00
MOVJ C00402 BC00402 VJ=20.00
'5.5.1
'------------------------
'W31.11
'------------------------
SFTON P0305
MOVL C00403 BC00403 V=333.3
MOVL C00404 BC00404 V=166.7 PL=0
MACRO1 MJ#(0) ARGF10
ARCON
MOVL C00405 BC00405 V=10.8
ARCOF
MOVL C00406 BC00406 V=166.7
SFTOF
'------------------------
'W31.13
'------------------------
SFTON P0306
MOVL C00407 BC00407 V=500.0
'SPR CZY W DOBRYM MIEJSCU SPOINA
MOVL C00408 BC00408 V=166.7 PL=0
ARCON
MOVL C00409 BC00409 V=10.8
ARCOF
MOVL C00410 BC00410 V=166.7
SFTOF
'------------------------
'W31.14
'------------------------
SFTON P0307
MOVL C00411 BC00411 V=333.3
MOVL C00412 BC00412 V=166.7 PL=0
ARCON
MOVL C00413 BC00413 V=8.3
ARCOF
MOVL C00414 BC00414 V=166.7
SFTOF
MOVL C00415 BC00415 V=333.3
MOVL C00416 BC00416 V=500.0
MOVJ C00417 BC00417 VJ=30.00
MOVJ C00418 BC00418 VJ=30.00
MOVJ C00419 BC00419 VJ=50.00
COMM '::::::::::::::::::::::::::::::::
COMM '::::::::::::::::::::::::::::::::
COMM '------------------------
COMM 'W27.9
COMM '------------------------
COMM '::::::::::::::::::::::::::::::::
COMM '::::::::::::::::::::::::::::::::
COMM MOVJ C00420 BC00420 VJ=25.00
COMM MOVJ C00421 BC00421 VJ=40.00
COMM SFTON P0404
COMM MOVL C00422 BC00422 V=500.0
COMM MOVL C00423 BC00423 V=166.7 PL=0
COMM MACRO1 MJ#(0) ARGF24
COMM ARCON
COMM MOVL C00424 BC00424 V=7.5
COMM ARCOF
COMM MOVL C00425 BC00425 V=166.7
COMM SFTOF
COMM '------------------------
COMM 'W27.11
COMM '------------------------
COMM SFTON P0406
COMM MOVL C00426 BC00426 V=666.7
COMM MOVL C00427 BC00427 V=166.7 PL=0
COMM MACRO1 MJ#(0) ARGF24
COMM ARCON
COMM MOVL C00428 BC00428 V=7.5
COMM ARCOF
COMM MOVL C00429 BC00429 V=166.7
COMM SFTOF
COMM '------------------------
COMM 'W27.13
'------------------------
COMM SFTON P0406
COMM MOVL C00430 BC00430 V=666.7
COMM MOVL C00431 BC00431 V=166.7 PL=0
COMM MACRO1 MJ#(0) ARGF24
COMM ARCON
COMM MOVL C00432 BC00432 V=7.5
COMM ARCOF
COMM MOVL C00433 BC00433 V=166.7
COMM SFTOF
COMM MOVJ C00434 BC00434 VJ=40.00
COMM MOVJ C00435 BC00435 VJ=50.00
COMM MOVJ C00436 BC00436 VJ=50.00
COMM MOVJ C00437 BC00437 VJ=50.00
MOVJ C00438 BC00438 VJ=50.00
'::::::::::::::::::::::::
'::::::::::::::::::::::::
'::::::::::::::::::::::::
'::::::::::::::::::::::::
'::::::::::::::::::::::::
'::::::::::::::::::::::::
'::::::::::::::::::::::::
MOVJ C00439 BC00439 VJ=50.00
MOVJ C00440 BC00440 VJ=50.00
'------------------------
'W214A
'------------------------
SFTON P0351
MOVL C00441 BC00441 V=500.0
MOVL C00442 BC00442 V=166.7 PL=0
MACRO1 MJ#(0) ARGF9
ARCON
SFTOF
SFTON P0350
MOVL C00443 BC00443 V=11.7
MOVL C00444 BC00444 V=11.0
ARCOF
MOVL C00445 BC00445 V=200.0
MOVL C00446 BC00446 V=333.3
SFTOF
MOVJ C00447 BC00447 VJ=50.00
MOVJ C00448 BC00448 VJ=50.00
MOVJ C00449 BC00449 VJ=50.00
MOVJ C00450 BC00450 VJ=40.00
MOVJ C00451 BC00451 VJ=50.00
MOVJ C00452 BC00452 VJ=30.00
MOVJ C00453 BC00453 VJ=30.00
MOVJ C00454 BC00454 VJ=30.00
MOVJ C00455 BC00455 VJ=30.00
'------------------------
'W31.16
'------------------------
SFTON P0308
MOVL C00456 BC00456 V=666.7
MOVL C00457 BC00457 V=166.7 PL=0
MACRO1 MJ#(0) ARGF10
ARCON
MOVL C00458 BC00458 V=10.8
ARCOF
MOVL C00459 BC00459 V=166.7
SFTOF
MOVL C00460 BC00460 V=666.7
MOVL C00461 BC00461 V=666.7
MOVL C00462 BC00462 V=666.7
MOVL C00463 BC00463 V=833.3
MOVL C00464 BC00464 V=666.7
MOVL C00465 BC00465 V=666.7
MOVL C00466 BC00466 V=333.3
MOVL C00467 BC00467 V=333.3
MOVL C00468 BC00468 V=250.0
MOVL C00469 BC00469 V=333.3
'------------------------
'W31.18
'------------------------
SFTON P0309
MOVL C00470 BC00470 V=166.7
MOVL C00471 BC00471 V=83.3 PL=0
ARCON
MOVL C00472 BC00472 V=10.8
ARCOF
MOVL C00473 BC00473 V=166.7
SFTOF
'------------------------
'W31.19
'------------------------
SFTON P0310
MOVL C00474 BC00474 V=333.3
MOVL C00475 BC00475 V=166.7 PL=0
ARCON
MOVL C00476 BC00476 V=10.8
ARCOF
MOVL C00477 BC00477 V=166.7
SFTOF
MOVL C00478 BC00478 V=333.3
MOVL C00479 BC00479 V=500.0
MOVL C00480 BC00480 V=666.7
MOVL C00481 BC00481 V=666.7
MOVJ C00482 BC00482 VJ=40.00
MOVJ C00483 BC00483 VJ=40.00
COMM '::::::::::::::::::::::::
COMM '::::::::::::::::::::::::
COMM '::::::::::::::::::::::::
COMM '::::::::::::::::::::::::
COMM '::::::::::::::::::::::::
COMM '::::::::::::::::::::::::
COMM '::::::::::::::::::::::::
COMM MOVJ C00484 BC00484 VJ=50.00
COMM MOVJ C00485 BC00485 VJ=30.00
COMM '::::::::::::::::::::::::::::::::
COMM '::::::::::::::::::::::::::::::::
COMM '------------------------
COMM 'W27.14
COMM '------------------------
COMM '::::::::::::::::::::::::::::::::
COMM '::::::::::::::::::::::::::::::::
COMM MOVL C00486 BC00486 V=500.0
COMM MOVL C00487 BC00487 V=500.0
COMM SFTON P0407
COMM MOVL C00488 BC00488 V=166.7 PL=0
COMM MACRO1 MJ#(0) ARGF24
COMM ARCON
COMM MOVL C00489 BC00489 V=7.5
COMM ARCOF
COMM MOVL C00490 BC00490 V=166.7
COMM SFTOF
COMM MOVJ C00491 BC00491 VJ=30.00
COMM '------------------------
COMM 'W27.16
COMM '------------------------
COMM SFTON P0408
COMM MOVL C00492 BC00492 V=500.0
COMM MOVL C00493 BC00493 V=166.7 PL=0
COMM MACRO1 MJ#(0) ARGF24
COMM ARCON
COMM MOVL C00494 BC00494 V=6.7
COMM ARCOF
COMM MOVL C00495 BC00495 V=166.7
COMM MOVL C00496 BC00496 V=666.7
COMM MOVJ C00497 BC00497 VJ=50.00
COMM SFTOF
COMM '------------------------
COMM 'W27.18
COMM '------------------------
COMM SFTON P0409
COMM MOVL C00498 BC00498 V=500.0
COMM MOVL C00499 BC00499 V=166.7 PL=0
COMM MACRO1 MJ#(0) ARGF24
COMM ARCON
COMM MOVL C00500 BC00500 V=7.5
COMM ARCOF
COMM MOVL C00501 BC00501 V=166.7
COMM SFTOF
COMM MOVJ C00502 BC00502 VJ=30.00
COMM MOVJ C00503 BC00503 VJ=30.00
COMM MOVJ C00504 BC00504 VJ=40.00
MOVJ C00505 BC00505 VJ=50.00
'::::::::::::::::::::::::
'::::::::::::::::::::::::
'::::::::::::::::::::::::
'::::::::::::::::::::::::
'::::::::::::::::::::::::
'::::::::::::::::::::::::
'::::::::::::::::::::::::
MOVJ C00506 BC00506 VJ=50.00
MOVJ C00507 BC00507 VJ=50.00
'------------------------
'W215A
'------------------------
SFTON P0359
MOVL C00508 BC00508 V=666.7
MOVL C00509 BC00509 V=166.7 PL=0
MACRO1 MJ#(0) ARGF9
ARCON
SFTOF
SFTON P0358
MOVL C00510 BC00510 V=11.7
ARCOF
MOVL C00511 BC00511 V=333.3
SFTOF
MOVJ C00512 BC00512 VJ=50.00
MOVJ C00513 BC00513 VJ=50.00
MOVJ C00514 BC00514 VJ=50.00
MOVJ C00515 BC00515 VJ=50.00
MOVJ C00516 BC00516 VJ=50.00
MOVJ C00517 BC00517 VJ=50.00
MOVJ C00518 BC00518 VJ=50.00
MOVL C00519 BC00519 V=500.0
'------------------------
'W31.21
'------------------------
SFTON P0311
MOVL C00520 BC00520 V=333.3
MOVL C00521 BC00521 V=166.7 PL=0
MACRO1 MJ#(0) ARGF10
ARCON
MOVL C00522 BC00522 V=10.8
ARCOF
MOVL C00523 BC00523 V=166.7
SFTOF
'------------------------
'W31.22
'------------------------
SFTON P0312
MOVL C00524 BC00524 V=666.7
MOVL C00525 BC00525 V=166.7 PL=0
ARCON
MOVL C00526 BC00526 V=10.8
ARCOF
MOVL C00527 BC00527 V=166.7
SFTOF
'------------------------
'W31.24
'------------------------
SFTON P0313
MOVL C00528 BC00528 V=666.7
MOVL C00529 BC00529 V=166.7 PL=0
ARCON
MOVL C00530 BC00530 V=10.8
ARCOF
MOVL C00531 BC00531 V=166.7
MOVL C00532 BC00532 V=166.7
MOVL C00533 BC00533 V=333.3
SFTOF
MOVL C00534 BC00534 V=333.3
MOVJ C00535 BC00535 VJ=30.00
MOVJ C00536 BC00536 VJ=30.00
MOVJ C00537 BC00537 VJ=50.00
MOVJ C00538 BC00538 VJ=50.00
COMM '::::::::::::::::::::::::
COMM '::::::::::::::::::::::::
COMM '::::::::::::::::::::::::
COMM '::::::::::::::::::::::::
COMM '::::::::::::::::::::::::
COMM '::::::::::::::::::::::::
COMM '::::::::::::::::::::::::
COMM MOVJ C00539 BC00539 VJ=50.00
COMM MOVJ C00540 BC00540 VJ=50.00
COMM '::::::::::::::::::::::::::::::::
COMM '::::::::::::::::::::::::::::::::
COMM '------------------------
COMM 'W27.19
COMM '------------------------
COMM '::::::::::::::::::::::::::::::::
COMM '::::::::::::::::::::::::::::::::
COMM MOVJ C00541 BC00541 VJ=30.00
COMM MOVL C00542 BC00542 V=666.7
COMM MOVL C00543 BC00543 V=250.0
COMM SFTON P0410
COMM MOVL C00544 BC00544 V=166.7 PL=0
COMM MACRO1 MJ#(0) ARGF24
COMM ARCON
COMM MOVL C00545 BC00545 V=7.5
COMM ARCOF
COMM MOVL C00546 BC00546 V=166.7
COMM SFTOF
COMM '------------------------
COMM 'W27.21
COMM '------------------------
COMM SFTON P0411
COMM MOVL C00547 BC00547 V=666.7
COMM MOVL C00548 BC00548 V=166.7 PL=0
COMM MACRO1 MJ#(0) ARGF24
COMM ARCON
COMM MOVL C00549 BC00549 V=7.5
COMM ARCOF
COMM MOVL C00550 BC00550 V=250.0
COMM SFTOF
COMM MOVJ C00551 BC00551 VJ=50.00
COMM MOVJ C00552 BC00552 VJ=50.00
COMM MOVJ C00553 BC00553 VJ=50.00
COMM '------------------------
COMM 'W27.22
COMM '------------------------
COMM MOVL C00554 BC00554 V=333.3
COMM MOVL C00555 BC00555 V=333.3
COMM SFTON P0412
COMM MOVL C00556 BC00556 V=166.7 PL=0
COMM MACRO1 MJ#(0) ARGF24
COMM ARCON
COMM MOVL C00557 BC00557 V=7.5
COMM ARCOF
COMM MOVL C00558 BC00558 V=200.0
COMM SFTOF
COMM '::::::::::::::::::::::::
COMM '::::::::::::::::::::::::
COMM '::::::::::::::::::::::::
COMM '::::::::::::::::::::::::
COMM '::::::::::::::::::::::::
COMM '::::::::::::::::::::::::
COMM '::::::::::::::::::::::::
COMM MOVJ C00559 BC00559 VJ=50.00
COMM MOVJ C00560 BC00560 VJ=50.00
COMM MOVJ C00561 BC00561 VJ=50.00
COMM MOVJ C00562 BC00562 VJ=50.00
MOVJ C00563 BC00563 VJ=50.00
'------------------------
'W215A
'------------------------
MOVJ C00564 BC00564 VJ=50.00
MOVJ C00565 BC00565 VJ=50.00
SFTON P0360
MOVL C00566 BC00566 V=500.0
MOVL C00567 BC00567 V=500.0
MOVL C00568 BC00568 V=166.7 PL=0
MACRO1 MJ#(0) ARGF9
ARCON
SFTOF
SFTON P0361
MOVL C00569 BC00569 V=11.7
MOVL C00570 BC00570 V=11.7
ARCOF
MOVL C00571 BC00571 V=500.0
SFTOF
MOVJ C00572 BC00572 VJ=50.00
MOVJ C00573 BC00573 VJ=50.00
MOVJ C00574 BC00574 VJ=50.00
MOVJ C00575 BC00575 VJ=80.00
MOVJ C00576 BC00576 VJ=50.00
MOVJ C00577 BC00577 VJ=50.00
MOVJ C00578 BC00578 VJ=40.00
MOVJ C00579 BC00579 VJ=20.00
MOVL C00580 BC00580 V=333.3
'------------------------
'W31.26
'------------------------
SFTON P0314
MOVL C00581 BC00581 V=833.3
MOVL C00582 BC00582 V=166.7 PL=0
MACRO1 MJ#(0) ARGF10
ARCON
MOVL C00583 BC00583 V=10.8
ARCOF
MOVL C00584 BC00584 V=200.0
SFTOF
'------------------------
'W31.27
'------------------------
SFTON P0316
MOVL C00585 BC00585 V=500.0
MOVL C00586 BC00586 V=166.7 PL=0
ARCON
MOVL C00587 BC00587 V=10.8
ARCOF
MOVL C00588 BC00588 V=200.0
SFTOF
MOVL C00589 BC00589 V=250.0
MOVL C00590 BC00590 V=250.0
MOVL C00591 BC00591 V=333.3
MOVL C00592 BC00592 V=416.7
MOVJ C00593 BC00593 VJ=30.00
MOVJ C00594 BC00594 VJ=50.00
MOVJ C00595 BC00595 VJ=50.00
COMM '::::::::::::::::::::::::
COMM '::::::::::::::::::::::::
COMM '::::::::::::::::::::::::
COMM '::::::::::::::::::::::::
COMM '::::::::::::::::::::::::
COMM '::::::::::::::::::::::::
COMM '::::::::::::::::::::::::
COMM MOVJ C00596 BC00596 VJ=50.00
COMM MOVJ C00597 BC00597 VJ=30.00
COMM MOVJ C00598 BC00598 VJ=30.00
COMM MOVJ C00599 BC00599 VJ=40.00
COMM MOVJ C00600 BC00600 VJ=50.00
COMM '::::::::::::::::::::::::::::::::
COMM '::::::::::::::::::::::::::::::::
COMM '------------------------
COMM 'W27.24
COMM '------------------------
COMM '::::::::::::::::::::::::::::::::
COMM '::::::::::::::::::::::::::::::::
COMM SFTON P0413
COMM MOVL C00601 BC00601 V=666.7
COMM MOVL C00602 BC00602 V=500.0
COMM MOVL C00603 BC00603 V=166.7 PL=0
COMM MACRO1 MJ#(0) ARGF24
COMM ARCON
COMM MOVL C00604 BC00604 V=7.5
COMM ARCOF
COMM MOVL C00605 BC00605 V=166.7
COMM SFTOF
COMM MOVJ C00606 BC00606 VJ=30.00
COMM MOVJ C00607 BC00607 VJ=30.00
COMM MOVJ C00608 BC00608 VJ=30.00
COMM '------------------------
COMM 'W27.26
COMM '------------------------
COMM SFTON P0414
COMM MOVL C00609 BC00609 V=333.3
COMM MOVL C00610 BC00610 V=333.3
COMM MOVL C00611 BC00611 V=166.7 PL=0
COMM MACRO1 MJ#(0) ARGF24
COMM ARCON
COMM MOVL C00612 BC00612 V=6.7
COMM ARCOF
COMM MOVL C00613 BC00613 V=200.0
SFTOF
COMM '------------------------
COMM 'W27.27
COMM '------------------------
COMM SFTON P0414
COMM MOVL C00614 BC00614 V=333.3
COMM MOVL C00615 BC00615 V=166.7 PL=0
COMM MACRO1 MJ#(0) ARGF24
COMM ARCON
COMM MOVL C00616 BC00616 V=6.7
COMM ARCOF
COMM MOVL C00617 BC00617 V=200.0
SFTOF
COMM MOVL C00618 BC00618 V=500.0
COMM '::::::::::::::::::::::::
COMM '::::::::::::::::::::::::
COMM '::::::::::::::::::::::::
COMM '::::::::::::::::::::::::
COMM '::::::::::::::::::::::::
COMM '::::::::::::::::::::::::
COMM '::::::::::::::::::::::::
COMM MOVL C00619 BC00619 V=833.3
COMM MOVJ C00620 BC00620 VJ=50.00
COMM MOVJ C00621 BC00621 VJ=50.00
COMM MOVJ C00622 BC00622 VJ=50.00
MOVJ C00623 BC00623 VJ=50.00
'------------------------
'W218A
'------------------------
MOVJ C00624 BC00624 VJ=50.00
MOVJ C00625 BC00625 VJ=50.00
SFTON P0357
MOVL C00626 BC00626 V=500.0
MOVL C00627 BC00627 V=500.0
MOVL C00628 BC00628 V=166.7 PL=0
MACRO1 MJ#(0) ARGF9
ARCON
SFTOF
SFTON P0356
MOVL C00629 BC00629 V=11.7
ARCOF
MOVL C00630 BC00630 V=333.3
SFTOF
MOVJ C00631 BC00631 VJ=50.00
MOVJ C00632 BC00632 VJ=50.00
MOVJ C00633 BC00633 VJ=50.00
MOVJ C00634 BC00634 VJ=50.00
MOVJ C00635 BC00635 VJ=50.00
MOVJ C00636 BC00636 VJ=50.00
MOVL C00637 BC00637 V=500.0
'------------------------
'W31.29
'------------------------
SFTON P0317
MOVL C00638 BC00638 V=333.3
MOVL C00639 BC00639 V=333.3
MOVL C00640 BC00640 V=166.7 PL=0
MOVL C00641 BC00641 V=166.7 PL=0
MACRO1 MJ#(0) ARGF10
ARCON
MOVL C00642 BC00642 V=10.8
ARCOF
MOVL C00643 BC00643 V=166.7
SFTOF
'------------------------
'W31.31
'------------------------
SFTON P0318
MOVL C00644 BC00644 V=666.7
MOVL C00645 BC00645 V=166.7 PL=0
MACRO1 MJ#(0) ARGF10
ARCON
MOVL C00646 BC00646 V=10.8
ARCOF
MOVL C00647 BC00647 V=200.0
MOVL C00648 BC00648 V=200.0
ARCON
MOVL C00649 BC00649 V=10.0
ARCOF
SFTOF
MOVL C00650 BC00650 V=200.0
MOVL C00651 BC00651 V=200.0
SFTOF
'------------------------
'W31.32
'------------------------
SFTON P0317
MOVL C00652 BC00652 V=166.7 PL=0
ARCON
MOVL C00653 BC00653 V=10.8
ARCOF
SFTOF
MOVL C00654 BC00654 V=333.3
MOVL C00655 BC00655 V=416.7
MOVL C00656 BC00656 V=500.0
MOVL C00657 BC00657 V=500.0
MOVL C00658 BC00658 V=500.0
MOVJ C00659 BC00659 VJ=40.00
MOVJ C00660 BC00660 VJ=50.00
MOVJ C00661 BC00661 VJ=50.00
COMM '::::::::::::::::::::::::
COMM '::::::::::::::::::::::::
COMM '::::::::::::::::::::::::
COMM '::::::::::::::::::::::::
COMM '::::::::::::::::::::::::
COMM '::::::::::::::::::::::::
COMM '::::::::::::::::::::::::
COMM MOVJ C00662 BC00662 VJ=50.00
COMM MOVJ C00663 BC00663 VJ=50.00
COMM MOVJ C00664 BC00664 VJ=30.00
COMM '::::::::::::::::::::::::::::::::
COMM '::::::::::::::::::::::::::::::::
COMM '------------------------
COMM 'W27.29
COMM '------------------------
COMM '::::::::::::::::::::::::::::::::
COMM '::::::::::::::::::::::::::::::::
COMM SFTON P0416
COMM MOVL C00665 BC00665 V=666.7
COMM MOVL C00666 BC00666 V=166.7 PL=0
COMM MACRO1 MJ#(0) ARGF24
COMM ARCON
COMM MOVL C00667 BC00667 V=6.7
COMM ARCOF
COMM MOVL C00668 BC00668 V=166.7
COMM SFTOF
COMM '------------------------
COMM 'W27.31
COMM '------------------------
COMM SFTON P0417
COMM MOVL C00669 BC00669 V=666.7
COMM MOVL C00670 BC00670 V=166.7
COMM ARCON
COMM MOVL C00671 BC00671 V=7.5
COMM ARCOF
COMM MOVL C00672 BC00672 V=250.0
COMM SFTOF
COMM '------------------------
COMM 'W27.32
COMM '------------------------
COMM '::::::::::::::::::::::::
COMM '::::::::::::::::::::::::
COMM '::::::::::::::::::::::::
COMM '::::::::::::::::::::::::
COMM '::::::::::::::::::::::::
COMM '::::::::::::::::::::::::
COMM '::::::::::::::::::::::::
COMM MOVL C00673 BC00673 V=666.7
COMM MOVJ C00674 BC00674 VJ=40.00
COMM MOVJ C00675 BC00675 VJ=40.00
COMM MOVJ C00676 BC00676 VJ=40.00
COMM MOVJ C00677 BC00677 VJ=40.00
COMM MOVJ C00678 BC00678 VJ=50.00
COMM '------------------------
COMM 'W219A
COMM '------------------------
MOVJ C00679 BC00679 VJ=50.00
MOVJ C00680 BC00680 VJ=50.00
SFTON P0353
MOVL C00681 BC00681 V=666.7
MOVL C00682 BC00682 V=250.0
MOVL C00683 BC00683 V=166.7 PL=0
MACRO1 MJ#(0) ARGF9
ARCON
SFTOF
SFTON P0352
MOVL C00684 BC00684 V=11.7
ARCOF
MOVL C00685 BC00685 V=250.0
SFTOF
MOVJ C00686 BC00686 VJ=50.00
MOVJ C00687 BC00687 VJ=50.00
CALL JOB:FRONT_WELD_-90ST-1_4840
CALL JOB:MOVE_OUT_OF_TUNNEL
END
